# B&R Automation Studio project Soiled_PLC (part 18)

#### 16_sdc3Cyclic.ab
```automation-basic
PROGRAM _CYCLIC
	(* cyclic program *)

;Sequence 16 - Discharger 3 D[916]

;-----------------------------------------
;Revision 1.00 19/12/2005 D.J. First Issue
;-----------------------------------------

DischargerEnable 		= (NOT Std.HaltSys)

I_BagAtBuffer			= FALSE
I_BagAtDischarger		= X[8].X07
I_OpenBag				= X[8].X08
I_LoadDropped			= X[8].X08
I_BagReleased			= FALSE
I_BagEmpty			  	= TRUE

I_BagAtEmptyBuffer		= FALSE ;X[11].X07
O_EmptyBagBufferOpen	= FALSE ;Y[11].Y07

O_BagReady				= FALSE
O_OpenBuffer 			= FALSE
O_Steadys				= FALSE
O_Closer				= FALSE
O_OpenBag				= FALSE
O_OpenStop				= FALSE

;Enable.SDC[1]			= FALSE
Request.SDC[3]			= FALSE

;Alarm
Alarm[16].Name 			= almNoAlarm ;Clear sequence alarm name
Alarm[16].Bag 			= 263
Alarm[16].Beacon		= TRUE
Alarm[16].Extra			= 0
Alarm[16].Time			= 3000

;Setup Sequence
STEP = D[916]
;Setup Pulse contact
PLS = (STEP <> LASTSTEP)
LASTSTEP = STEP

;Step 0 - Disabled
IF (STEP = 0) THEN
	;Disabled
ENDIF

;Check Status - Bag settled at buffer, no bag at discharger, bag at buffer on screen and no bag at discharger on the screen
TON_10ms(I_BagAtBuffer,300,SettledAtBuffer,SettledAtBufferET)
IF (STEP = 1) THEN
	;IF (DischargerEnable AND SettledAtBuffer AND NOT I_BagAtDischarger AND (Bag[261].Cat > 0) AND (Bag[263].Cat = 0) AND NOT Std.HaltSys) THEN
	IF (DischargerEnable AND NOT I_BagAtDischarger AND (Bag[263].Cat = 0) AND NOT Std.HaltSys) THEN
		D[916] = 2
	ENDIF
	IF (Bag[263].Cat > 0) THEN
		Alarm[16].Name = almBagDataError
	ELSE IF I_BagAtDischarger THEN
		Alarm[16].Name = almSwitchFault
	;ELSE IF (Bag[263].Cat > 0) AND NOT I_BagAtBuffer THEN
	;	Alarm[16].Name 	= almBagDataError
	;	Alarm[16].Bag	= 263
	;ELSE IF (Bag[261].Cat = 0) AND I_BagAtBuffer THEN
	;	Alarm[16].Name 	= almBagNotShownOnScreen
	;	Alarm[16].Bag	= 261
	ENDIF
ENDIF

;Wait for bag in discharger
IF (STEP = 2) THEN
	;Enable.SDC[1]	= TRUE
	;O_OpenBuffer 	= TRUE
	IF I_BagAtDischarger THEN
		D[916] = 3
	ENDIF
	;Alarm[16].Name = almBagNotArrived
ENDIF

;Let bag settle in discharger
TON_10ms(((STEP = 3) AND I_BagAtDischarger),1000,SettledAtDischarger,SettledAtDischargerET)
IF (STEP = 3) THEN
	IF PLS  AND (Bag[263].Cat = 0) AND (Bag[252].Cat > 0) THEN
		Bag[252].Dst = 0
		Bag[263]     = Bag[252]
		Bag[252]     = Bag[0]
	ENDIF
	IF SettledAtDischarger THEN
		D[916] = 4
	ENDIF
	IF (Bag[263].Cat = Std.MaxCats) THEN
		D[916] = 11
	ENDIF
	Alarm[16].Name = almBagNotSettled
ENDIF

;Allow steadys to move down
TON_10ms((STEP = 4),400,SteadysDown,SteadysDownET)
IF (STEP = 4) THEN
	IF (SteadysDown AND NOT I_OpenBag) THEN
		D[916] = 5
	ENDIF
	IF I_OpenBag THEN
		Alarm[16].Name = almSwitchFault
	ENDIF
ENDIF

;Steady cylinders on from steps 4 - 9
O_Steadys = ((STEP >= 4) AND (STEP <= 9))

;Bag opener on from step 5 - 8
O_OpenBag = ((STEP >= 6) AND (STEP <= 8))

;Bag Ready to Washing Machine
IF (STEP = 5) THEN
	O_BagReady = TRUE
	IF I_OpenBag OR TestDischarger THEN
		D[916] = 6
	ENDIF
ENDIF

;Set LoadDropped to False
IF (STEP <> 6) THEN
	LoadDropped = FALSE
ENDIF

;Open Bag Until LoadDropped recieved and has been open for 6 seconds
TON_10ms((STEP = 6),600,MinOpen,MinOpenET) ;ET means Elapsed Time
IF (STEP = 6) THEN

	IF NOT I_OpenBag OR TestDischarger THEN
	;IF I_BagEmpty THEN
		LoadDropped = TRUE
	ENDIF

	IF (LoadDropped AND MinOpen) THEN
		;Write Report
		;------------
		IF (ReportUnloading[3].Cat = 0) THEN
			ReportUnloading[3].Cat = UINT(Bag[263].Cat)	;Category
			ReportUnloading[3].Cus = Bag[263].Cus		;Customer
			ReportUnloading[3].Wgt = Bag[263].Wgt		;Weight
			ReportUnloading[3].Cnt = 0					;Count
			ReportUnloading[3].Stn = 0					;Station
			ReportUnloading[3].Mcn = 3					;Machine
		ENDIF
	ENDIF
	IF (LoadDropped AND MinOpen) THEN
		D[916] = 7
	ENDIF
	Alarm[16].Name = almLoadNotDropped
ENDIF

;Change display to empty bag
IF (STEP = 7) THEN
	O_BagReady = Std.Clock500ms
	IF (I_OpenBag OR TestDrop) THEN
		Bag[263].Cat 	= Std.MaxCats
		D[916] 			= 8
	ENDIF
	Alarm[16].Name = almGeneralSequence
ENDIF

;Close bag
TON_10ms((STEP = 8),700,CloserDown,CloserDownET)
IF (STEP = 8) THEN
	O_Closer = TRUE
	IF CloserDown THEN
		D[916] = 9
	ENDIF
ENDIF

;Allow closer to go back up
TON_10ms((STEP = 9),700,CloserUp,CloserUpET)
IF (STEP = 9) THEN
	IF CloserUp THEN
		D[916] = 10
	ENDIF
ENDIF

;Allow steadys to go up
TON_10ms((STEP = 10),400,SteadyUp,SteadyUpET)
IF (STEP = 10) THEN
	IF SteadyUp THEN
		D[916] = 11
	ENDIF
ENDIF

;Check for space on empty bag buffer
IF (STEP = 11) THEN
	Request.SDC[3] = TRUE
	IF Enable.SDC[3] THEN
		D[916] = 12
	ENDIF
ENDIF

;Open buffer stop - unitl bag out
IF (STEP = 12) THEN
	O_OpenStop 	= TRUE
	Bag[263] 	= Bag[0]
	IF NOT Enable.SDC[3] THEN
		D[916] = 1
	ENDIF
	Alarm[16].Name = almBagNotReleased
ENDIF

;Alarms
TimerAlarm.IN 	= NOT PLS AND (Alarm[16].Name > 0)
TimerAlarm.PT 	= Alarm[16].Time
TimerAlarm FUB TON_10ms()
Alarm[16].On 	= TimerAlarm.Q
Alarm[16].ET 	= TimerAlarm.ET

;Outputs
Y[8].Y08 	= O_BagReady
;Y[6].Y01 	= O_OpenBuffer
Y[8].Y09 	= O_Steadys
Y[8].Y10 	= O_OpenBag
Y[8].Y05 	= O_Closer
Y[8].Y11 	= O_OpenStop
END_PROGRAM
```

### Program Logical/ExportsFromOriginal/17_svc2 (IEC, version 1.00.0) - * SVC2 Vertical Conveyor

#### 17_svc2Cyclic.ab
```automation-basic
PROGRAM _CYCLIC
	(* cyclic program *)

;---------------------------------------------------
;Sequence 13 - SIC2 Soiled Incline Conveyor 2 D[913]
;---------------------------------------------------

;Inputs
I_CarriageAtTop         = X[5].X02
I_CarriageAtBottom      = X[5].X03
I_BagOutAtTopSVC2       = X[7].X07
I_BagOutAtBottom		= X[4].X16
I_BagOnCarriageSVC2 	= X[5].X04
I_BagAtSVCBuffer        = X[6].X01

O_OpenCarriageStop		= FALSE
O_MoveUp 				= FALSE
O_MoveDown              = FALSE
O_BufferStop            = FALSE

Request.SVC[2] 			= FALSE

Alarm[17].Name 			= 0
Alarm[17].Bag			= 250
Alarm[17].Beacon		= TRUE
Alarm[17].Extra			= 0
Alarm[17].Time			= 3000

;Setup Sequence
STEP = D[917]
;Setup Pulse contact
PLS = (STEP <> LASTSTEP)
LASTSTEP = STEP

;Sequence
;Step 0 - Disabled
IF (STEP = 0) THEN
	;Disabled
ENDIF

;Move carriage up
IF (STEP = 1) THEN
	O_MoveUp = TRUE
	IF I_CarriageAtTop THEN
		D[917] = 2
	ENDIF
	IF NOT Std.EStop THEN
		Alarm[17].Name = almCarriageMoveFault
	ENDIF
ENDIF

;check carriage

IF (STEP = 2) THEN
	IF (NOT I_BagOnCarriageSVC2 AND NOT I_BagOutAtTopSVC2 AND  (Bag[250].Cat = 0) AND NOT Std.HaltSys) THEN

		D[917] = 3
	ENDIF
	IF (Bag[250].Cat > 0)  THEN
		Alarm[17].Name 	= almBagDataError
		Alarm[17].Bag	= 250
	ELSE IF  I_BagOnCarriage THEN
		Alarm[17].Name 	= almSwitchFault
		Alarm[17].Bag	= 250
	ENDIF
ENDIF

;request a bag
IF (STEP = 3) THEN
	;Request.SVC[2]  	= (I_CarriageAtTop AND NOT I_BagOnCarriageSVC2)
ENDIF

;Request a bag
TON_10ms(I_BagAtSVCBuffer AND (Bag[230].Cat > 0),200,BagAtBuffer,BagAtBufferET)
IF (STEP = 3) THEN

	IF (BagAtBuffer AND (Bag[230].Dst = 23) and (Bag[252].Cat = 0) and (Bag[263].Cat = 0) AND (D[916] = 2)) THEN
		D[917] = 4
	ELSE IF BagAtBuffer AND (Bag[230].Dst < 23) THEN
		D[917] = 4
	ENDIF

ENDIF

;wait for bag to arrive

IF (STEP = 4) THEN
	O_BufferStop  = TRUE

	IF (Bag[230].Dst = 23) AND I_CarriageAtTop   THEN
		O_OpenCarriageStop = TRUE
	ENDIF

	IF I_BagOutAtTopSVC2 AND O_OpenCarriageStop THEN
		IF((Bag[230].Cat > 0 ) AND (Bag[252].Cat = 0)) THEN
			Bag[252] = Bag[230]
			Bag[230] = Bag[0]
		ENDIF
		D[917] = 1
	ELSE IF ((Bag[230].Dst < 23) AND (Bag[230].Cat > 0)) THEN
		IF I_BagOnCarriageSVC2 THEN
			IF((Bag[230].Cat > 0 ) AND (Bag[250].Cat = 0)) THEN
				Bag[250] = Bag[230]
				Bag[230] = Bag[0]
			ENDIF
			D[917] = 5
		ENDIF

	ENDIF
ENDIF

;Allow bag to settle
TON_10ms(((STEP = 5) AND I_BagOnCarriageSVC2),300,BagSettled,BagSettledET)
IF (STEP = 5) THEN

	IF BagSettled THEN
		D[917] = 6
	ENDIF
	Alarm[17].Name = almBagNotSettled
ENDIF

;check bottom roller switch
IF (STEP = 6) THEN
	IF NOT I_CarriageAtBottom THEN
		D[917] = 7
	ENDIF
ENDIF

;move carriage down
IF (STEP = 7) THEN
	O_MoveDown 		= TRUE
	IF I_CarriageAtBottom THEN
		D[917] = 8
	ENDIF
ENDIF

;Check buffer has space
IF (STEP = 8) THEN
	IF Line[25].Clear AND (Bag[251].Cat = 0) AND (Bag[258].Cat = 0) AND NOT I_BagOutAtBottom THEN
		C[16] = 0
		C[25] = 0
		D[917] = 9
	ENDIF
	IF (Bag[258].Cat = 0) AND NOT Line[25].Clear THEN
		Alarm[17].Name = almBagNotSettled
		Alarm[17].Bag  = 258
	ENDIF
ENDIF

;Release bag low level

IF (STEP = 9) THEN
	O_OpenCarriageStop		= TRUE
	IF PLS THEN
		C[16] = 0
	ENDIF
	IF Line[16].Clear AND NOT PLS AND Carrstoptimer THEN
		IF ((Bag[250].Cat > 0) AND (Bag[251].Cat = 0)) THEN
			Bag[251] = Bag[250]
			Bag[250] = Bag[0]
		ENDIF
		D[917] = 10
	ENDIF
	Alarm[17].Name = almBagNotReleased
	Alarm[17].Bag  = 250
ENDIF
TON_10ms(((STEP = 9) AND O_OpenCarriageStop),750,Carrstoptimer,CarrstoptimerET)

;Bag at buffer stop high level
IF (STEP = 10) THEN
	IF BagAtBuffer THEN
		D[917] = 1
	ENDIF
ENDIF

;move trans bag to buffer
IF Line[25].Trip THEN
	IF ((Bag[251].Cat > 0) AND (Bag[258].Cat = 0)) THEN
		Bag[258] = Bag[251]
		Bag[251] = Bag[0]
	ENDIF
ENDIF

;Alarms
TimerAlarm.IN 	= NOT PLS AND (Alarm[17].Name > 0)
TimerAlarm.PT 	= Alarm[17].Time
TimerAlarm FUB TON_10ms()
Alarm[17].On 	= TimerAlarm.Q
Alarm[17].ET 	= TimerAlarm.ET

;Outputs

Y[9].Y03 =  (O_OpenCarriageStop	AND (I_CarriageAtTop OR I_CarriageAtBottom))
Y[9].Y01 =  (O_MoveUp AND NOT I_CarriageAtTop)
Y[9].Y02 =  (O_MoveDown AND NOT I_CarriageAtBottom)
Y[6].Y01 =  (O_BufferStop AND I_CarriageAtTop)
END_PROGRAM
```

#### 17_svc2.var
```iecst
VAR RETAIN
	STEP	:UINT;
	PLS	:BOOL;
	LASTSTEP	:UINT;
	O_OpenBufferStop	:BOOL;
	I_BagAtBuffer	:BOOL;
	O_RunMotor	:BOOL;
	BagSettled	:BOOL;
	BagSettledET	:TIME;
	BagAtBuffer	:BOOL;
	RunOnET	:TIME;
	RunOn	:BOOL;
	BagNearTopET	:TIME;
	BagNearTop	:BOOL;
	BagAtBufferET	:UDINT;
	I_BagInIncline	:BOOL;
END_VAR

VAR
	I_BagAtOutgoingBuffer	:BOOL;
	I_PaddleInPosition	:BOOL;
	CloseBufferStop	:BOOL;
	CloseBufferStopET	:TIME;
	O_OutgoingBufferOpen	:BOOL;
	TimerAlarm	:TON_10ms;
	O_SelectSP4ToSP2	:BOOL;
	I_BagReleased	:BOOL;
	O_SelectSP4	:BOOL;
	I_BagOutAtTop	:BOOL;
	I_BagOutAtBottom	:BOOL;
	I_BagOnCarriage	:BOOL;
	I_CarriageAtTop	:BOOL;
	I_CarriageAtBottom	:BOOL;
	O_OpenCarriageStop	:BOOL;
	O_MoveUp	:BOOL;
	O_MoveDown	:BOOL;
	I_BagAtSVCBuffer	:BOOL;
	O_BufferStop	:BOOL;
	Carrstoptimer	:BOOL;
	CarrstoptimerET	:TIME;
END_VAR
```

- Visualisation Logical/ExportsFromOriginal/svc1 (not shown)

### Data object Logical/ExportsFromOriginal/can_cmd (Simple) - * Powertrans 1 & 2

#### can_cmd.dat
```
;-----------------
;CAN Command Table
;-----------------

;         1234567890123456789012345678901   1234567890123456789012345678901
00000121,"ReadFrame1                     ","EventRead1                     ",$00000000
00000120,"WriteFrame1                    ","EventWrite1                    ",$00000001

00000131,"ReadFrame2                     ","EventRead2                     ",$00000000
00000130,"WriteFrame2                    ","EventWrite2                    ",$00000001

;00000141,"ReadFrame3                     ","EventRead3                     ",$00000000
;00000140,"WriteFrame3                    ","EventWrite3                    ",$00000001
;   |          |                                 |                               |
; CAN ADR  Variable Name 31 Chrs             Event Variable 31 Chrs           Read = 0 Write = 1
```

### Program Logical/ExportsFromOriginal/can_drv2 (IEC, version 1.00.0) - * PowerTrans 1 SDC2

#### can_drv2Cyclic.ab
```automation-basic
PROGRAM _CYCLIC
;----------------------------------------
;Version 1.00 08/02/2005 D.J. First Issue
;----------------------------------------

IF CANOK THEN

	;----------------
	;Set Write values
	;----------------

	;Powertrans 1
	IF CAN[1].BagReady THEN
		WriteFrame1.ControlSignals = BIT_SET(WriteFrame1.ControlSignals, 1)
	ELSE
		WriteFrame1.ControlSignals = BIT_CLR(WriteFrame1.ControlSignals, 1)
	ENDIF
	;IF CAN[1].DoubleLoad THEN
	;	WriteFrame1.ControlSignals = BIT_SET(WriteFrame1.ControlSignals, 2)
	;ELSE
	;	WriteFrame1.ControlSignals = BIT_CLR(WriteFrame1.ControlSignals, 2)
	;ENDIF
	WriteFrame1.Destination = 0
	WriteFrame1.Category 	= CAN[1].Category
	WriteFrame1.Customer    = CAN[1].Customer
	WriteFrame1.Weight      = CAN[1].Weight

	;Write to Machine1
	EventWrite1 = TRUE

	;Powertrans 2
	IF CAN[2].BagReady THEN
		WriteFrame2.ControlSignals = BIT_SET(WriteFrame2.ControlSignals, 1)
	ELSE
		WriteFrame2.ControlSignals = BIT_CLR(WriteFrame2.ControlSignals, 1)
	ENDIF
	;IF CAN[2].DoubleLoad THEN
	;	WriteFrame2.ControlSignals = BIT_SET(WriteFrame2.ControlSignals, 2)
	;ELSE
	;	WriteFrame2.ControlSignals = BIT_CLR(WriteFrame2.ControlSignals, 2)
	;ENDIF
	WriteFrame2.Destination = 0
	WriteFrame2.Category 	= CAN[2].Category
	WriteFrame2.Customer    = CAN[2].Customer
	WriteFrame2.Weight      = CAN[2].Weight

	;Write to Machine2
	EventWrite2 = TRUE

	;-----------------
	;Service CAN table
	;-----------------

	IF CANdftab_01.status=0 THEN						(*check error level*)
		CANrwtab_01.enable		= 1
		CANrwtab_01.tab_ident	= CANdftab_01.tab_ident (*define tab_id*)
		CANrwtab_01 FUB CANrwtab()						(*initiate CANrwtab*)
		LastError = CANrwtab_01.status
	ENDIF

	;----------------------------------
	;Check for incomming data from CBW1
	;----------------------------------

	;Powertrans 1
	IF EventRead1 THEN

		EventRead1 = FALSE

		CAN[1].Live 		  = BIT_TST(ReadFrame1.ControlSignals,0)
		CAN[1].DropLoad 	  = BIT_TST(ReadFrame1.ControlSignals,1)
		CAN[1].LoadDropped    = BIT_TST(ReadFrame1.ControlSignals,2)

		IF CAN[1].Live THEN
			CAN[1].LiveTime = 50	;5 seconds
		ENDIF

	ENDIF

	;----------------------------------
	;Check for incomming data from CBW2
	;----------------------------------

	;Powertrans 2
	IF EventRead2 THEN

		EventRead2 = FALSE

		CAN[2].Live 		  = BIT_TST(ReadFrame2.ControlSignals,0)
		CAN[2].DropLoad 	  = BIT_TST(ReadFrame2.ControlSignals,1)
		CAN[2].LoadDropped    = BIT_TST(ReadFrame2.ControlSignals,2)

		IF CAN[2].Live THEN
			CAN[2].LiveTime = 50	;5 seconds
		ENDIF

	ENDIF

	;-------------------
	;CAN Live / Presence
	;-------------------

	LOOP n = 1 TO 2 DO

		IF (CAN[n].LiveTime > 0) THEN
			CAN[n].LiveTime = (CAN[n].LiveTime - 1)
		ENDIF

		CAN[n].Live = (CAN[n].LiveTime <> 0)

	ENDLOOP

ENDIF
END_PROGRAM
```

#### can_drv2Init.ab
```automation-basic
PROGRAM _INIT
	(* init program *)

CAN_enable = 1
EventWrite1 = 0									;Reset CAN data table WRITE event
EventRead1 = 0  								;Reset CAN data table READ event
;EventWrite2 = 0								;Reset CAN data table WRITE event
;EventRead2 = 0  								;Reset CAN data table READ event
;EventWrite3 = 0								;Reset CAN data table WRITE event
;EventRead3 = 0  							    ;Reset CAN data table READ event

CANopen_01.enable		= CAN_enable
CANopen_01.baud_rate	= 25					;Define baud rate - 250 kbit/s
CANopen_01.cob_anz		= 100      				;Define number of link objects
CANopen_01.error_adr	= ADR(error_var)		;Define address for error output
CANopen_01.device		= ADR("SS1.IF2")	;Define number of device
CANopen_01.info			= 0

CANopen_01 FUB CANopen()						;Initiate CANopen

IF CANopen_01.status=0 THEN						;Check error level

	DOInfo.enable = 1
	DOInfo.pName  = "can_cmd"

	DOInfo FUB DatObjInfo()

	IF (DOInfo.status = 0) THEN

		data_adr					= DOInfo.pDatObjMem
		CANdftab_01.enable			= 1
		CANdftab_01.us_ident 		= CANopen_01.us_ident	;Set us_id
		CANdftab_01.table_adr		= data_adr				;Define address of data object
		CANdftab_01.tab_num			= UINT(DOInfo.len / 72)	;Define number of values

		CANdftab_01 FUB CANdftab()    						;Initiate CANdftab

		IF CANdftab_01.status = 0 THEN
			WriteFrame1.ControlSignals = BIT_SET(WriteFrame1.ControlSignals,0);Set Live Signal
			WriteFrame2.ControlSignals = BIT_SET(WriteFrame2.ControlSignals,0)
			;WriteFrame3.ControlSignals = BIT_SET(WriteFrame3.ControlSignals,0)
			CANOK = TRUE
		ENDIF

	ENDIF

ENDIF
END_PROGRAM
```

#### can_drv2.var
```iecst
VAR RETAIN
	CAN_enable	:BOOL;
	ReadFrame1	:WET_CAN;
	EventRead1	:BOOL;
	EventWrite1	:BOOL;
	LastError	:UINT;
	n	:UINT;
	CANOK	:BOOL;
	WriteFrame1	:WET_CAN;
	EventWrite2	:BOOL;
END_VAR

VAR
	ReadFrame2	:WET_CAN;
	EventRead2	:BOOL;
	WriteFrame2	:WET_CAN;
	CANopen_01	:CANopen;
	DOInfo	:DatObjInfo;
	CANdftab_01	:CANdftab;
	error_var	:UDINT;
	data_adr	:UDINT;
	CANrwtab_01	:CANrwtab;
END_VAR
```

### Program Logical/ExportsFromOriginal/can_dis (IEC, version 1.00.0)

#### can_disCyclic.ab
```automation-basic
PROGRAM _CYCLIC
;-----------------------------------------
;Revision 1.00 18/02/2002 D.J. First Issue
;-----------------------------------------

;2 * 20 or 2 * 40 chr VFD display

;Set D register where text for display is set E register for weight
DisplayChrs		= 80

LOOP m = 1 TO 16 DO
	DisplayCat[m] = (4000 + ((m - 1) * 80))
	DisplayCus[m] = DisplayCat[m] + 40
	DisplayWgt[m] = Bag[200 + m].Wgt
ENDLOOP

LOOP x = 1 to 16 DO

	memcpy(ADR(Display[0]) ,ADR(D[DisplayCat[x]]),DisplayChrs)
	memcpy(ADR(Display[44]),ADR(D[DisplayCus[x]]),DisplayChrs)

	;As the weight value is a INT put into a UINT -0.1 = 65535
	;Display only if less than 500kg
	IF (DisplayWgt[x] < 5000) THEN
		DIS4(DisplayWgt[x],TRUE,Dummy,Wgt1s,Wgt10s,Dummy)
	ELSE
		Wgt1s 	= 0
		Wgt10s 	= 0
	ENDIF

	;Add Weight and goto next line
	Display[35] = $20 ;Space
	Display[36] = (48 + USINT(Wgt10s))
	Display[37] = (48 + USINT(Wgt1s))
	Display[38] = $6B 	;k
	Display[39] = $67 	;g
	Display[40] = $A	;Line Feed
	Display[41] = $D	;Carriage Return
	Display[42] = 0
	Display[43] = 0

	;Display[78] = $44	;D
	;Display[79] = $55	;U
	;Display[80] = $43	;C
	;Display[81] = $4B	;K
	;Display[82] = $45	;E
	;Display[83] = $52	;R

	;Cursor Off and Home
	IF (STEP = 0) THEN
		n = 0
		Data.Data[0] = $9B
		Data.Data[1] = $6C
		Data.Data[2] = $9B
		Data.Data[3] = $48
		Data.Data[4] = 0
		Data.Data[5] = 0
		Data.Data[6] = 0
		Data.Data[7] = 0
	ENDIF

	;Write text to the Display
	IF (STEP > 0) THEN
		Data.Data[0] = USINT(Display[0 + n])
		Data.Data[1] = USINT(Display[1 + n])
		Data.Data[2] = USINT(Display[2 + n])
		Data.Data[3] = USINT(Display[3 + n])
		Data.Data[4] = USINT(Display[4 + n])
		Data.Data[5] = USINT(Display[5 + n])
		Data.Data[6] = USINT(Display[6 + n])
		Data.Data[7] = USINT(Display[7 + n])
	ENDIF

	;Write to the CAN Frame For the Current Display
	IF (x = 1) THEN
		DisplayTXFrame1 = Data
	ELSE IF (x = 2) THEN
		DisplayTXFrame2 = Data
	ELSE IF (x = 3) THEN
		DisplayTXFrame3 = Data
	ELSE IF (x = 4) THEN
		DisplayTXFrame4 = Data
	ELSE IF (x = 5) THEN
		DisplayTXFrame5 = Data
	ELSE IF (x = 6) THEN
		DisplayTXFrame6 = Data
	ELSE IF (x = 7) THEN
		DisplayTXFrame7 = Data
	ELSE IF (x = 8) THEN
		DisplayTXFrame8 = Data
	ELSE IF (x = 9) THEN
		DisplayTXFrame9 = Data
	ELSE IF (x = 10) THEN
		DisplayTXFrame10 = Data
	ELSE IF (x = 11) THEN
		DisplayTXFrame11 = Data
	ELSE IF (x = 12) THEN
		DisplayTXFrame12 = Data
	ELSE IF (x = 13) THEN
		DisplayTXFrame13 = Data
	ELSE IF (x = 14) THEN
		DisplayTXFrame14 = Data
	ELSE IF (x = 15) THEN
		DisplayTXFrame15 = Data
	ELSE IF (x = 16) THEN
		DisplayTXFrame16 = Data
	ENDIF

ENDLOOP

IF (STEP > 0) THEN
	n = n + 8
ENDIF

STEP = STEP + 1

StepsRequired = ((DisplayChrs / 8) + 1) ;Steps = Total Chrs / 8 + 1
IF STEP > StepsRequired THEN
	STEP = 0
ENDIF

IF CANOK THEN

	;------------------------------------------------------
	;Configure the CAN write to CBW1 SDC1
	;------------------------------------------------------

	;Write to Displays
	DisplayWrite1 = TRUE
	;DisplayWrite2 = TRUE
	DisplayWrite3 = TRUE
	;DisplayWrite4 = TRUE
	DisplayWrite5 = TRUE
	;DisplayWrite6 = TRUE
	DisplayWrite7 = TRUE
	;DisplayWrite8 = TRUE
	;DisplayWrite9 = TRUE
	;DisplayWrite10 = TRUE
	;DisplayWrite11 = TRUE
	;DisplayWrite12 = TRUE
	;DisplayWrite13 = TRUE
	;DisplayWrite14 = TRUE
	;DisplayWrite15 = TRUE
	;DisplayWrite16 = TRUE

	;------------------------
	;Service CAN table
	;------------------------

	IF CANdftab_01.status=0 THEN						(*check error level*)
		CANrwtab_01.enable		= 1
		CANrwtab_01.tab_ident	= CANdftab_01.tab_ident (*define tab_id*)
		CANrwtab_01 FUB CANrwtab()						(*initiate CANrwtab*)
		LastError = CANrwtab_01.status
	ENDIF

	;-----------------
	;Read Display Data
	;-----------------
	IF DisplayRead1 THEN
		DisplayRead1 = FALSE
		Reply = DisplayRXFrame1.Data[1]
	ENDIF
	IF DisplayRead2 THEN
		DisplayRead2 = FALSE
		Reply = DisplayRXFrame2.Data[1]
	ENDIF
	IF DisplayRead3 THEN
		DisplayRead3 = FALSE
		Reply = DisplayRXFrame3.Data[1]
	ENDIF
	IF DisplayRead4 THEN
		DisplayRead4 = FALSE
		Reply = DisplayRXFrame4.Data[1]
	ENDIF
	IF DisplayRead5 THEN
		DisplayRead5 = FALSE
		Reply = DisplayRXFrame5.Data[1]
	ENDIF
	IF DisplayRead6 THEN
		DisplayRead6 = FALSE
		Reply = DisplayRXFrame6.Data[1]
	ENDIF
	IF DisplayRead7 THEN
		DisplayRead7 = FALSE
		Reply = DisplayRXFrame7.Data[1]
	ENDIF
	IF DisplayRead8 THEN
		DisplayRead8 = FALSE
		Reply = DisplayRXFrame8.Data[1]
	ENDIF
	IF DisplayRead9 THEN
		DisplayRead9 = FALSE
		Reply = DisplayRXFrame9.Data[1]
	ENDIF
	IF DisplayRead10 THEN
		DisplayRead10 = FALSE
		Reply = DisplayRXFrame10.Data[1]
	ENDIF
	IF DisplayRead11 THEN
		DisplayRead11 = FALSE
		Reply = DisplayRXFrame11.Data[1]
	ENDIF
	IF DisplayRead12 THEN
		DisplayRead12 = FALSE
		Reply = DisplayRXFrame12.Data[1]
	ENDIF
	IF DisplayRead13 THEN
		DisplayRead13 = FALSE
		Reply = DisplayRXFrame13.Data[1]
	ENDIF
	IF DisplayRead14 THEN
		DisplayRead14 = FALSE
		Reply = DisplayRXFrame14.Data[1]
	ENDIF
	IF DisplayRead15 THEN
		DisplayRead15 = FALSE
		Reply = DisplayRXFrame15.Data[1]
	ENDIF
	IF DisplayRead16 THEN
		DisplayRead16 = FALSE
		Reply = DisplayRXFrame16.Data[1]
	ENDIF

ENDIF
END_PROGRAM
```

#### can_disInit.ab
```automation-basic
PROGRAM _INIT
	(* init program *)

CAN_enable = 1
DisplayWrite1 = 0								;Reset CAN data table WRITE event
DisplayRead1 = 0  								;Reset CAN data table READ event
;EventWrite2 = 0								;Reset CAN data table WRITE event
;EventRead2 = 0  								;Reset CAN data table READ event
;EventWrite3 = 0								;Reset CAN data table WRITE event
;EventRead3 = 0  							    ;Reset CAN data table READ event

CANopen_01.enable		= CAN_enable
CANopen_01.baud_rate	= 25					;Define baud rate - 250 kbit/s
CANopen_01.cob_anz		= 100      				;Define number of link objects
CANopen_01.error_adr	= ADR(error_var)		;Define address for error output
CANopen_01.device		= ADR("SS1.IF3")		;Define number of device
CANopen_01.info			= 0

CANopen_01 FUB CANopen()						;Initiate CANopen

IF CANopen_01.status=0 THEN						;Check error level

	DOInfo.enable = 1
	DOInfo.pName  = "disp_cmd"

	DOInfo FUB DatObjInfo()

	IF (DOInfo.status = 0) THEN

		data_adr					= DOInfo.pDatObjMem
		CANdftab_01.enable			= 1
		CANdftab_01.us_ident 		= CANopen_01.us_ident	;Set us_id
		CANdftab_01.table_adr		= data_adr				;Define address of data object
		CANdftab_01.tab_num			= UINT(DOInfo.len / 72)	;Define number of values

		CANdftab_01 FUB CANdftab()    						;Initiate CANdftab

		IF CANdftab_01.status = 0 THEN
			CANOK = TRUE
		ENDIF

	ENDIF

ENDIF
END_PROGRAM
```

#### can_dis.var
```iecst
VAR RETAIN
	CAN_enable	:BOOL;
	LastError	:UINT;
	n	:UINT;
	CANOK	:BOOL;
END_VAR

VAR
	CANopen_01	:CANopen;
	DOInfo	:DatObjInfo;
	CANdftab_01	:CANdftab;
	error_var	:UDINT;
	data_adr	:UDINT;
	CANrwtab_01	:CANrwtab;
	DisplayWrite1	:BOOL;
	DisplayRead1	:BOOL;
	DisplayCat	:ARRAY [0..16] OF UINT;
	DisplayWgt	:ARRAY [0..12] OF UINT;
	DisplayCus	:ARRAY [0..16] OF UINT;
	Display	:ARRAY [0..87] OF UINT;
	Data	:WriteDisplay;
	Reply	:USINT;
	DisplayRXFrame5	:ReadDisplay;
	DisplayRXFrame4	:ReadDisplay;
	DisplayWrite4	:BOOL;
	DisplayTXFrame1	:WriteDisplay;
	DisplayWrite5	:BOOL;
	DisplayTXFrame2	:WriteDisplay;
	x	:UINT;
	DisplayWrite6	:BOOL;
	DisplayTXFrame3	:WriteDisplay;
	DisplayRead2	:BOOL;
	DisplayTXFrame4	:WriteDisplay;
	DisplayRead3	:BOOL;
	DisplayTXFrame5	:WriteDisplay;
	Dummy	:UINT;
	DisplayRead4	:BOOL;
	DisplayRXFrame1	:ReadDisplay;
	DisplayTXFrame6	:WriteDisplay;
	DisplayRead5	:BOOL;
	DisplayRXFrame2	:ReadDisplay;
	DisplayRead6	:BOOL;
	DisplayRXFrame3	:ReadDisplay;
	StepsRequired	:UINT;
	DisplayChrs	:UINT;
	DisplayRXFrame6	:ReadDisplay;
	STEP	:UINT;
	Wgt1s	:UINT;
	DisplayWrite2	:BOOL;
	DisplayWrite3	:BOOL;
	Wgt10s	:UINT;
	m	:UINT;
	DisplayTXFrame7	:WriteDisplay;
	DisplayTXFrame8	:WriteDisplay;
	DisplayTXFrame9	:WriteDisplay;
	DisplayTXFrame10	:WriteDisplay;
	DisplayTXFrame11	:WriteDisplay;
	DisplayTXFrame12	:WriteDisplay;
	DisplayTXFrame13	:WriteDisplay;
	DisplayWrite7	:BOOL;
	DisplayWrite8	:BOOL;
	DisplayWrite9	:BOOL;
	DisplayWrite10	:BOOL;
	DisplayWrite11	:BOOL;
	DisplayWrite12	:BOOL;
	DisplayWrite13	:BOOL;
	DisplayWrite14	:BOOL;
	DisplayWrite15	:BOOL;
	DisplayWrite16	:BOOL;
	DisplayRead7	:BOOL;
	DisplayRead8	:BOOL;
	DisplayRead9	:BOOL;
	DisplayRead10	:BOOL;
	DisplayRead11	:BOOL;
	DisplayRead12	:BOOL;
	DisplayRead13	:BOOL;
	DisplayRead14	:BOOL;
	DisplayRead15	:BOOL;
	DisplayRead16	:BOOL;
	DisplayRXFrame7	:ReadDisplay;
	DisplayRXFrame8	:ReadDisplay;
	DisplayRXFrame9	:ReadDisplay;
	DisplayRXFrame10	:ReadDisplay;
	DisplayRXFrame11	:ReadDisplay;
	DisplayRXFrame12	:ReadDisplay;
	DisplayRXFrame13	:ReadDisplay;
	DisplayRXFrame14	:ReadDisplay;
	DisplayRXFrame15	:ReadDisplay;
	DisplayRXFrame16	:ReadDisplay;
	DisplayTXFrame14	:WriteDisplay;
	DisplayTXFrame15	:WriteDisplay;
	DisplayTXFrame16	:WriteDisplay;
END_VAR
```

### Data object Logical/ExportsFromOriginal/disp_cmd (Simple, version 1.00.0)

#### disp_cmd.dat
```
;-----------------
;CAN Command Table
;-----------------

;         1234567890123456789012345678901   1234567890123456789012345678901
;CAN Node 11
00001215,"DisplayRXFrame1                ","DisplayRead1                   ",$00000000
00001214,"DisplayTXFrame1                ","DisplayWrite1                  ",$00000001
;CAN Node 12
;00001231,"DisplayRXFrame2                ","DisplayRead2                   ",$00000000
;00001230,"DisplayTXFrame2                ","DisplayWrite2                  ",$00000001
;CAN Node 13
00001247,"DisplayRXFrame3                ","DisplayRead3                   ",$00000000
00001246,"DisplayTXFrame3                ","DisplayWrite3                  ",$00000001
;CAN Node 14
;00001263,"DisplayRXFrame4                ","DisplayRead4                   ",$00000000
;00001262,"DisplayTXFrame4                ","DisplayWrite4                  ",$00000001
;CAN Node 15
00001279,"DisplayRXFrame5                ","DisplayRead5                   ",$00000000
00001278,"DisplayTXFrame5                ","DisplayWrite5                  ",$00000001
;CAN Node 16
;00001295,"DisplayRXFrame6                ","DisplayRead6                   ",$00000000
;00001294,"DisplayTXFrame6                ","DisplayWrite6                  ",$00000001
;CAN Node 17
00001311,"DisplayRXFrame7                ","DisplayRead7                   ",$00000000
00001310,"DisplayTXFrame7                ","DisplayWrite7                  ",$00000001
;CAN Node 18
;00001327,"DisplayRXFrame8                ","DisplayRead8                   ",$00000000
;00001326,"DisplayTXFrame8                ","DisplayWrite8                  ",$00000001
;CAN Node 19
;00001343,"DisplayRXFrame9                ","DisplayRead9                   ",$00000000
;00001342,"DisplayTXFrame9                ","DisplayWrite9                  ",$00000001
;CAN Node 20
;00001359,"DisplayRXFrame10               ","DisplayRead10                  ",$00000000
;00001358,"DisplayTXFrame10               ","DisplayWrite10                 ",$00000001
;CAN Node 21
;00001375,"DisplayRXFrame11               ","DisplayRead11                  ",$00000000
;00001374,"DisplayTXFrame11               ","DisplayWrite11                 ",$00000001
;CAN Node 22
;00001391,"DisplayRXFrame12               ","DisplayRead12                  ",$00000000
;00001390,"DisplayTXFrame12               ","DisplayWrite12                 ",$00000001
;CAN Node 23
;00001407,"DisplayRXFrame13               ","DisplayRead13                  ",$00000000
;00001406,"DisplayTXFrame13               ","DisplayWrite13                 ",$00000001
;CAN Node 24
;00001423,"DisplayRXFrame14               ","DisplayRead14                  ",$00000000
;00001422,"DisplayTXFrame14               ","DisplayWrite14                 ",$00000001
;CAN Node 25
;00001439,"DisplayRXFrame15               ","DisplayRead15                  ",$00000000
;00001438,"DisplayTXFrame15               ","DisplayWrite15                 ",$00000001
;CAN Node 26
;00001455,"DisplayRXFrame16               ","DisplayRead16                  ",$00000000
;00001454,"DisplayTXFrame16               ","DisplayWrite16                 ",$00000001

;   |          |                                 |                               |
; CAN ADR  Variable Name 31 Chrs             Event Variable 31 Chrs           Read = 0 Write = 1
```

### Safety.typ
```iecst
TYPE
	SafeInterlockType : 	STRUCT
		GS_DI_01_Access_Reset : BOOL; (*Interlock access request and zone reset operator input*)
		GS_DI_02_Monitor_Solenoid : BOOL; (*Interlock solenoid feedback*)
		GS_DO_01_Lock_Solenoid : BOOL; (*Interlock solenoid output*)
		GS_Two_Channel_Input : BOOL; (*Safe PLC feedback of the state of interlock dual channel*)
	END_STRUCT;
	SafeE_StopType : 	STRUCT
		ES_SI_Two_Channel : ARRAY[0..MAX_DUAL_CHANNELS]OF BOOL; (*Safe PLC feedback of the state of e-stop dual channel*)
	END_STRUCT;
	SafeTowerLightType : 	STRUCT
		TL_DO_Green : BOOL; (*Tower light output for Green light*)
		TL_DO_Yellow : BOOL; (*Tower light output for Yellow light*)
		TL_DO_Red : BOOL; (*Tower light output for Red light*)
		TL_DO_Sounder : BOOL; (*Tower light output for sounder*)
	END_STRUCT;
	SafeZoneType : 	STRUCT
		Interlock : SafeInterlockType; (*Interlock structure*)
		E_Stop : SafeE_StopType; (*Emergency stop structure*)
		TowerLight : SafeTowerLightType; (*Tower light structure*)
		Zone_Status : BOOL; (*State of the zone passed back from safe PLC*)
		AccessRequested : BOOL; (*Operator as requested access*)
		BagsInTransit : BOOL; (*True = Sequences are still not in a safe step*)
		HoistsOutOfPosition : BOOL; (*True = Hoists in zone are not parked*)
		Main_Reset : BOOL; (*Main panel reset*)
		Main_Lamp : BOOL; (*Main panel lamp*)
		Disable : BOOL; (*Passed into sequences to inhibit stepping on*)
		EDM : BOOL; (*EDM Feedback from linking relays*)
		ResetReady : BOOL; (*Zone is ready to be reset*)
		LiftGates : BOOL; (*Lift the edge protection gates.*)
	END_STRUCT;
	Safety_Hoist_type : 	STRUCT
		I_Operator_PushButton : BOOL; (*Bulk loading operator push button*)
		O_OpenGuard : BOOL; (*Sliding guard output*)
		O_CloseGuard : BOOL; (*Sliding guard output*)
		OutOfPosition : BOOL; (*True when hoist is not in Service position*)
		I_GuardClosed : BOOL; (*Sliding guard closed*)
	END_STRUCT;
END_TYPE
```

### Safety.var
```iecst
VAR
	SafetyZone : ARRAY[0..MAX_SAFE_ZONES] OF SafeZoneType;
	Safety_Master_Reset : BOOL;
	Safety_Module_Fault : BOOL;
	Hoist_Safety : ARRAY[0..MAX_HOIST] OF Safety_Hoist_type;
END_VAR
VAR CONSTANT
	MAX_SAFE_ZONES : USINT := 3;
	MAX_DUAL_CHANNELS : USINT := 1;
	MAX_HOIST : USINT := 1;
END_VAR
```

### Program Logical/Safety/Safety (IEC, version 1.00.4)

#### Main.st - Safet Task must come after all task with gaurded areas
```iecst
//---------------------------------------------
//-------------Safety Request------------------
//---------------------------------------------
//V1.00.2 -- 2019 May 24 -- TR -- Fix issue with master reset not working if not ready.
//V1.00.3 -- 2019 June 26 -- TR -- FIx issue with the solenoid not opening if the hoist switch is made after the bagInTransit timers.. Add timer for hoist in position so the hoist cannot be moving past the safe position and open the door.
//V1.00.4 -- 2019 November 11 -- TR -- 	FIX: Issues with the solenoid locking incorrectly,
										//ADD: Control to lift the edge protection gates ( Map Directly to all required outputs.)
PROGRAM _INIT
debounceMasterPT := 200; //2 second
transitSettlePT := 3000; //3000seconds
startUpWarningPT := 500; //5 secs
enableMasterReset := TRUE; // Set to true if master reset is to be used
FOR n:=0 TO MAX_SAFE_ZONES DO
	safeState[n] := 4;
END_FOR;
END_PROGRAM

PROGRAM _CYCLIC

ton_10ms_startUp_Warning(IN:=ton_10ms_Master_Reset.Q, PT:=startUpWarningPT);
Safety_Master_Reset := ton_10ms_startUp_Warning.Q AND Std.Clock1s;

IF SafetyZone[0].Main_Reset AND enableMasterReset THEN
	masterResetRequest := 1; // Set masterResetRequest
END_IF;
ton_10ms_Master_Reset(IN:= masterResetRequest, PT:=debounceMasterPT);

FOR n:=0 TO MAX_SAFE_ZONES DO
	//-------------------------------------------------------
	//---------------------Master-reset----------------------
	//-------------------------------------------------------

	lockDoor[n] := FALSE;

	tof_HoistsOutOfPosition[n].IN := SafetyZone[n].HoistsOutOfPosition;
	tof_HoistsOutOfPosition[n].PT := 100;
	tof_HoistsOutOfPosition[n]();

	ton_entryError[n].IN := (safeState[n] = 3);
	ton_entryError[n].PT := 100;
	ton_entryError[n]();

	IF ton_10ms_Master_Reset.Q AND NOT SafetyZone[n].Zone_Status AND SafetyZone[n].ResetReady THEN // only put a zone to reset if it needs it
		masterReset[n] := TRUE; // Set masterReset
		safeState[n] := 10; // Goto master reset state
	END_IF;

	//-------------------------------------------------------
	//------------------END-Master-Reset-END-----------------
	//-------------------------------------------------------

	//-------------------------------------------------------
	//------------------Safety-State-Machine-----------------
	//-------------------------------------------------------

	//Wait for bags to finish moving and hoists to get into position.. Door can be unlocked
	ton_10ms_Transit_Settle[n](IN:=SafetyZone[n].AccessRequested AND (safeState[n] = 1), PT:=transitSettlePT);
	f_trigRequestAccess[n].CLK:= SafetyZone[n].Interlock.GS_DI_01_Access_Reset;
	f_trigRequestAccess[n]();
	CASE safeState[n] OF
		0: //Zone reset do not enter

			// Operator requests access by pressing Access DI for 1 second then releasing
			//ton_10ms_Access_Debounce[n](IN:=SafetyZone[n].Interlock.GS_DI_01_Access_Reset, PT:=debouncePT);
			//Request Access on f_trig of pressing reset. if the zone is healthy
			//SafetyZone[n].Interlock.GS_DO_01_Lock_Solenoid := FALSE; //Reset after reset pressed and door shut
			IF SafetyZone[n].Zone_Status AND f_trigRequestAccess[n].Q  THEN//	ELSIF (debounceEdgeNeg[n] OR SafetyZone[n].AccessRequested) AND NOT masterReset THEN //Look for falling edge if masterReset not requested
				SafetyZone[n].AccessRequested := TRUE; //Reset after unlocking or safe zone goes off
				safeState[n] := 1; //Access has been requested
				masterReset[n] := 0;
				//If zone accessed by override or depedant Zone drops out.
			ELSIF NOT SafetyZone[n].Zone_Status AND NOT SafetyZone[n].Interlock.GS_Two_Channel_Input THEN //If entered with overide goto state 3
				safeState[n] := 3;
			ELSIF NOT SafetyZone[n].Zone_Status AND SafetyZone[n].Interlock.GS_Two_Channel_Input THEN //If dependant zone drops out
				safeState[n] := 4;
			END_IF;

		1: //Access has been requested
			//Allow 1 second for moving bags to settle, once ok
			ton_10ms_bagsInTransit[n](IN:=NOT SafetyZone[n].BagsInTransit, PT:=100); //buffer the BagsInTransit bool

			//Latch solenoid lock open
			IF ton_10ms_bagsInTransit[n].Q AND SafetyZone[n].Disable AND NOT tof_HoistsOutOfPosition[n].Q THEN //Use Disable instead of AccessRequested, to ensure one cyclic check with Disable on to stop BagsInTransit being missed
				//SafetyZone[n].Interlock.GS_DO_01_Lock_Solenoid := TRUE; //Reset after reset pressed and door shut
				safeState[n] := 2; //Safe to enter no bags in transit
			ELSIF ton_10ms_Transit_Settle[n].Q THEN
				//SafetyZone[n].Interlock.GS_DO_01_Lock_Solenoid := NOT tof_HoistsOutOfPosition[n].Q; //Reset after reset pressed and door shut
				safeState[n] := 3; //Waiting time elapsed, enter with caution
			END_IF;

			//If zone accessed by override or depedant Zone drops out.
			IF NOT SafetyZone[n].Zone_Status AND NOT SafetyZone[n].Interlock.GS_Two_Channel_Input THEN //If entered with overide goto state 3
				safeState[n] := 3;
			ELSIF NOT SafetyZone[n].Zone_Status AND SafetyZone[n].Interlock.GS_Two_Channel_Input THEN //If dependant zone drops out
				safeState[n] := 4;
			ELSIF SafetyZone[n].Zone_Status AND f_trigRequestAccess[n].Q THEN //Cancel the request
				SafetyZone[n].AccessRequested := FALSE; //Reset after safe zone goes off
				safeState[n] := 4;
			END_IF;

		2..3: //Zone unlocked
			//Reset access request
			lockDoor[n] := NOT tof_HoistsOutOfPosition[n].Q;

			IF SafetyZone[n].AccessRequested AND NOT SafetyZone[n].Zone_Status THEN
				SafetyZone[n].AccessRequested := FALSE; //Reset after safe zone goes off
				IF n = 0 THEN
					safeState[n] := 0; //Zone reset do not enter
				END_IF
			ELSIF SafetyZone[n].Zone_Status AND f_trigRequestAccess[n].Q  AND SafetyZone[n].AccessRequested THEN //Cancel the request
				SafetyZone[n].AccessRequested := FALSE; //Reset after safe zone goes off
				safeState[n] := 4;
			ELSIF SafetyZone[n].Zone_Status AND NOT SafetyZone[n].AccessRequested THEN // zone has been accessed and reset.
				safeState[n] := 0;
			END_IF;

		4:
			//Reset tower light state only if safety plc feedback ok
			IF SafetyZone[n].Zone_Status THEN //Check Safe PLC status
				safeState[n] := 0; //Zone reset do not enter
			END_IF;

		10: // Master reset
			IF (SafetyZone[n].Zone_Status OR NOT SafetyZone[n].ResetReady) THEN
				safeState[n] := 0;
				masterReset[n] := FALSE;
			END_IF;

	END_CASE;

//	//Lock solenoid
//	//ton_10ms_Reset_Debounce[n](IN:=SafetyZone[n].Interlock.GS_DI_01_Access_Reset, PT:=debouncePT);
//	IF (SafetyZone[n].Interlock.GS_DI_01_Access_Reset AND (safeState[n] > 1) AND NOT masterReset[n]) THEN
//		//SafetyZone[n].Interlock.GS_DO_01_Lock_Solenoid := FALSE; //Reset after reset pressed and door shut
//		SafetyZone[n].AccessRequested := FALSE;
//		safeState[n] := 4; // Check zone status
//		//		ELSIF masterReset AND NOT SafetyZone[n].Zone_Status AND SafetyZone[n].ResetReady THEN
//		//			safeState[n] := 10; // Goto master reset state
//	END_IF;

	//Set disable to safe zone off or access requested
	SafetyZone[n].Disable := SafetyZone[n].AccessRequested OR NOT SafetyZone[n].Zone_Status;

	//-------------------------------------------------------
	//-------END--------Safety State Machine-------END-------
	//-------------------------------------------------------

	//-------------------------------------------------------
	//---------Set tower light status-&-TV-Indicators--------
	//-------------------------------------------------------
	IF (n > 0) THEN //Light tower 0 does not need to indicate access state.. It is used on the main cab to indicate alarms. See alarm Task.
		SafetyZone[n].TowerLight.TL_DO_Green := SafetyZone[n].TowerLight.TL_DO_Yellow := SafetyZone[n].TowerLight.TL_DO_Red := SafetyZone[n].TowerLight.TL_DO_Sounder := 0;
		CASE safeState[n] OF
			0: //Zone reset do not enter
				SafetyZone[n].TowerLight.TL_DO_Green 	:= SafetyZone[n].Zone_Status;
				SafetyZone[n].TowerLight.TL_DO_Red 		:= NOT SafetyZone[n].Zone_Status;
			1: //Access has been requested
				SafetyZone[n].TowerLight.TL_DO_Yellow 	:= Std.Clock1s; 	//Means Zone Ok but access requested
				SafetyZone[n].TowerLight.TL_DO_Green 	:= SafetyZone[n].Zone_Status;
				SafetyZone[n].TowerLight.TL_DO_Red 		:= NOT SafetyZone[n].Zone_Status;
			2: //Safe to enter no bags in transit and hoists in position
				SafetyZone[n].TowerLight.TL_DO_Yellow 	:= TRUE; //Amber & RED steady indicates safe to enter
				SafetyZone[n].TowerLight.TL_DO_Green 	:= SafetyZone[n].Zone_Status;
				SafetyZone[n].TowerLight.TL_DO_Red 		:= TRUE;
			3: //
				SafetyZone[n].TowerLight.TL_DO_Yellow 	:= Std.Clock200ms; //Amber/Green Alternate-- Enter with Caution
				SafetyZone[n].TowerLight.TL_DO_Sounder 	:= NOT ton_entryError[n].Q; //Short alarm to indicate enter with caution
				SafetyZone[n].TowerLight.TL_DO_Green 	:= NOT Std.Clock200ms;
			SafetyZone[n].TowerLight.TL_DO_Red 		:= NOT Std.Clock200ms OR SafetyZone[n].HoistsOutOfPosition; // If red ight on then fault

			4: //Ready for Reset
				SafetyZone[n].TowerLight.TL_DO_Yellow 	:= Std.Clock500ms AND SafetyZone[n].ResetReady; //Flash Yellow when ready to be reset
				SafetyZone[n].TowerLight.TL_DO_Green 	:= SafetyZone[n].Zone_Status;

			10://Master Reset Zone about to start
				SafetyZone[n].TowerLight.TL_DO_Sounder := TRUE;
				SafetyZone[n].TowerLight.TL_DO_Red := Std.Clock200ms; //Red fast flash indicates zone will reset

		END_CASE;

	END_IF;

	//-------------------------------------------------------------
	//-------END-Set tower light status-&-TV-Indicators-END--------
	//-------------------------------------------------------------

	//Check if the master reset has reset all zones.
	IF (masterReset[n] AND NOT SafetyZone[n].Zone_Status) THEN
		resetRequired := 1;
	END_IF;

	SafetyZone[n].Interlock.GS_DO_01_Lock_Solenoid := lockDoor[n];
	SafetyZone[n].LiftGates := (SafetyZone[n].Zone_Status AND (SafetyZone[n].BagsInTransit OR NOT SafetyZone[n].AccessRequested)); // Edge protection gates.

END_FOR;

IF NOT resetRequired THEN
	masterResetRequest := 0;
END_IF;
resetRequired := 0;

//Flash reset btn on main cabinet
IF masterResetRequest THEN // We can do a master reset and not out safe 0 to reset
	SafetyZone[0].Main_Lamp := Std.Clock200ms;
ELSE
	SafetyZone[0].Main_Lamp := Std.Clock1s AND NOT SafetyZone[0].Zone_Status;
END_IF;

//--------------------CUSTOMISTATION FOR INDICATION--------------------

//FOR n := 0 TO MAX_DUAL_CHANNELS DO
//	Indication[40 + n] := NOT SafetyZone[0].E_Stop.ES_SI_Two_Channel[n];
//END_FOR;
//
//Indication[61]	:= NOT SafetyZone[1].Interlock.GS_Two_Channel_Input;
//Indication[62]	:= NOT SafetyZone[2].Interlock.GS_Two_Channel_Input;
//Indication[63] 	:= NOT SafetyZone[3].Interlock.GS_Two_Channel_Input;
//Indication[64] 	:= NOT SafetyZone[4].Interlock.GS_Two_Channel_Input;
//
////Fire Doors
//Indication[65] 	:= NOT SafetyZone[1].E_Stop.ES_SI_Two_Channel[1];
//Indication[66] 	:= NOT SafetyZone[1].E_Stop.ES_SI_Two_Channel[2];

END_PROGRAM
```

#### Variables.var - Local variables
```iecst
VAR
	n : UINT;
	transitSettlePT : UDINT; (*Determines the amount of time to wait for bags in transit to settle before opening the interlock*)
	ton_10ms_Transit_Settle : ARRAY[0..MAX_SAFE_ZONES] OF TON_10ms; (*Determines the amount of time to wait for bags in transit to settle before opening the interlock*)
	safeState : ARRAY[0..MAX_SAFE_ZONES] OF USINT; (*USINT that tracks the state of the safe system so it can control the tower light*)
	debounceMasterPT : UDINT;
	masterReset : ARRAY[0..MAX_SAFE_ZONES] OF BOOL;
	ton_10ms_Master_Reset : TON_10ms;
	masterResetRequest : BOOL;
	startUpWarningPT : UDINT;
	ton_10ms_startUp_Warning : TON_10ms;
	tp_10ms_reset_Pulse : TP_10ms;
	enableMasterReset : BOOL;
	ton_10ms_Reset_Debounce : ARRAY[0..MAX_SAFE_ZONES] OF TON_10ms;
	ton_10ms_bagsInTransit : ARRAY[0..MAX_SAFE_ZONES] OF TON_10ms;
	f_trigRequestAccess : ARRAY[0..MAX_SAFE_ZONES] OF F_TRIG;
	ton_entryError : ARRAY[0..MAX_SAFE_ZONES] OF TON_10ms;
	resetRequired : BOOL;
	lockDoor : ARRAY[0..MAX_SAFE_ZONES] OF BOOL;
	tof_HoistsOutOfPosition : ARRAY[0..MAX_SAFE_ZONES] OF TOF_10ms;
END_VAR
```

### Program Logical/Safety/AccessControl (IEC) - *Mapping to allow access into zones

#### Main.st
```iecst
PROGRAM _CYCLIC

//	Std.SafetyOnZone[1]	;SPC1
//	Std.SafetyOnZone[2]	;SVC1
//	Std.SafetyOnZone[3]	;SVC2/3

//No access on zone 0

	SafetyZone[0].BagsInTransit :=  FALSE;  // Safe to enter when false (Switch is NO) FALSE WHEN OK..
	SafetyZone[0].HoistsOutOfPosition := FALSE; //<-- This is used to stop the door from opening if not position FALSE IS OK -- SWITCH IS NC..

	SafetyZone[1].BagsInTransit :=  FALSE;
	SafetyZone[1].HoistsOutOfPosition := FALSE;
//
	SafetyZone[2].BagsInTransit :=  FALSE;
	SafetyZone[2].HoistsOutOfPosition := Hoist_Safety[1].OutOfPosition;// OR Hoist_Safety[7].OutOfPosition;
//
	SafetyZone[3].BagsInTransit :=  FALSE;
	SafetyZone[3].HoistsOutOfPosition := FALSE;///Hoist_Safety[1].OutOfPosition OR Hoist_Safety[2].OutOfPosition OR Hoist_Safety[3].OutOfPosition;

END_PROGRAM
```

### Program Logical/Safety/SafetyUI (IEC) - Handling

#### SafetyUI.st - Implementation code
```iecst
(********************************************************************
* COPYRIGHT -- Bernecker + Rainer
********************************************************************
* Program: SafetySample
* File: SafetySample.st
* Author: B&R
********************************************************************
* Implementation of program SafetySample
********************************************************************)

PROGRAM _INIT

(* command structure for remote control FUB *)
	remotecmd.Version := safeVERSION_R107;	(* version *)
	remotecmd.Password := 'safeplc';				(* password *)
	remotecmd.NewPassword 	:= 'safeplc';

	remoteCmdGetStatus 		:= remotecmd;
	remoteCmdGetStatus.Command		:= safeCMD_STATUS;
	remoteCmdGetStatus.Data			:= 0;
	remoteCmdGetStatus.Number := 10;// ID to show request from auto refresh

	remoteControlcmd ACCESS ADR(remoteCmdGetStatus);

	(* command structure for application download *)
	appcmd1.Version := safeVERSION_R107;	(* version *)
	appcmd1.Password := 'safeplc';					(* password *)
	appcmd1.ApplicationID := 1;				(* application id *)

//	(* command structure for machine options download *)
//	datacmd1.Version := safeVERSION_R107;								(* version *)
//	datacmd1.Password := '';											(* password *)
//	datacmd1.pDeviceListInput := ADR(visuDeviceListInput);				(* device list *)
//	datacmd1.pMachineOptionsInput := ADR(dataMachineOptionsBitInput);	(* bit machine options *)
//	datacmd1.pModuleFlagsInput := ADR(dataModuleFlagsInput);			(* module flags *)
//	datacmd1.pAcknMachineOptions := ADR(dataAcknMachineOptions);		(* acknowledge information *)

//	(* command structure for extended machine options *)
//	datacmd2.Version := safeVERSION_R107;					(* version *)
//	datacmd2.Password := '';								(* password *)
//	datacmd2.pIntDataInput := ADR(visuIntInput);			(* INT channels *)
//	datacmd2.NumberIntInput := 1;							(* number of INT channels *)
//	datacmd2.pUintDataInput := ADR(visuUintInput);			(* UINT channels *)
//	datacmd2.NumberUintInput := 1;							(* number of UINT channels *)
//	datacmd2.pDintDataInput := ADR(visuDintInput);			(* DINT channels *)
//	datacmd2.NumberDintInput := 1;							(* number of DINT channels *)
//	datacmd2.pUdintDataInput := ADR(visuUdintInput);		(* UDINT channels *)
//	datacmd2.NumberUdintInput := 1;							(* number of UDINT channels *)
//	datacmd2.pAcknMachineOptions := ADR(visuAcknExtData);	(* acknowledge information *)

	(* hide elements in visualization *)
	FOR xcnt := 0 TO SIZEOF(statusButtonActiv) - 1 DO
		statusButtonActiv[xcnt] := 1;
	END_FOR

	(* hide elements in visualization *)
	statusButtonUnlockApp := 1;
	statusButtonUnlockData := 1;
	statusAcknInfoData := 1;
	statusButtonUnlockExtData := 1;
	statusAcknInfoExtData := 1;
	statusDialog := 1;

	(* set SafeLOGIC ID *)
	visuUsedSLIDRemote := 1;
	visuUsedSLIDData := 1;

	slxused := 1;
	safety := 0;
	visuEnableButtons := 0;

END_PROGRAM

PROGRAM _CYCLIC

//on init make sure we have set the password..

	ton_refreshStatus(IN := (safety > 0) AND SafetyPLC_Ok AND NOT safeRemoteControl_0.Busy AND NOT ton_refreshStatus.Q, PT:=100);

//	//Alarm for Hoist
//	IF (safeLogicStatus.SafeOSState <> 16#66) THEN //16# is Run[SAFE]
//		MpAlarmXSet(gAlarmXCore_Link,'SafetyPLCNotRunning');
//	ELSIF EDGEPOS(safeLogicStatus.SafeOSState = 16#66) THEN
//		MpAlarmXReset(gAlarmXCore_Link,'SafetyPLCNotRunning');
//	END_IF;
//	//End of Alarm

	CASE safety OF
		0: // Set the password on app load
			visuEnableButtons := 0;
			IF SafetyPLC_Ok THEN
				remotecmd.Command 	:= safeCMD_ENTER;
				remotecmd.Number 	:= 0;
				remotecmd.Data		:= safeCMD_SK_PW;
				IF safeRemoteControl_0.Done THEN
					safety := 10;
				ELSIF EDGEPOS(safeRemoteControl_0.Error) THEN
					execute := 0;
				END_IF;
				safeRemoteControl_0(SafeLOGICID := visuUsedSLIDRemote, Execute := execute, pCommandData := ADR(remotecmd));
				execute := 1;
			END_IF;

		10:// RUN UI

			//Lock the control buttons when the fub's are busy.
			visuEnableButtons := SafetyPLC_Ok AND ((remoteControlcmd.Number = 10) OR NOT safeRemoteControl_0.Busy) AND NOT safeDownloadApplication_0.Busy;
			(****************************************************************************************************************************************)
			(****************************************************************************************************************************************)
			(****************************************************************************************************************************************)
			(* show dialog to ackn command *)
			IF (dialogRemoteCmd = 1) THEN
				statusDialog := 0;
				dialogRemoteCmd := 0;
				indexButtonLeft := 0;
				indexButtonRight := 1;
				indexHeaderText := 0;
				IF (remotecmd.Data = safeCMD_SK_FORMAT) THEN
					indexMessageText := 0;
				ELSIF (remotecmd.Data = safeCMD_SK_XCHG) THEN
					indexMessageText := 1;
				ELSIF (remotecmd.Data = safeCMD_1_UDID_ACKN) THEN
					indexMessageText := 2;
				ELSIF (remotecmd.Data = safeCMD_2_UDID_ACKN) THEN
					indexMessageText := 3;
				ELSIF (remotecmd.Data = safeCMD_3_UDID_ACKN) THEN
					indexMessageText := 4;
				ELSIF (remotecmd.Data = safeCMD_4_UDID_ACKN) THEN
					indexMessageText := 5;
				ELSIF (remotecmd.Data =  safeCMD_N_UDID_ACKN) THEN
					indexMessageText := 6;
				ELSIF (remotecmd.Data =  safeCMD_CLEAR_DATA) THEN
					indexMessageText := 7;
				ELSIF (remotecmd.Data = safeCMD_FW_ACKN) THEN
					indexMessageText := 8;
				ELSIF (remotecmd.Data = safeCMD_RESET) THEN
					indexMessageText := 9;
				END_IF
			END_IF

			(* if dialog is ackn execute fub *)
			IF (dialogButtonLeft = 1 AND indexHeaderText = 0) THEN
				executeRemoteCmd := 1;
				dialogButtonLeft := 0;
				statusDialog := 1;
			ELSIF (dialogButtonRight = 1 AND indexHeaderText = 0) THEN
				dialogButtonRight := 0;
				statusDialog := 1;
			END_IF

			(* password must be at least 6 characters long *)
			IF brsstrlen(ADR(remotecmd.NewPassword)) < 6 THEN
				statusSetPassword := 2;
			ELSE
				statusSetPassword := 0;
			END_IF

			IF NOT safeRemoteControl_0.Busy THEN
				IF executeRemoteCmd THEN
					remoteControlcmd ACCESS ADR(remotecmd);
					executeRemoteControl := 1;
					executeRemoteCmd := 0;
				ELSIF ton_refreshStatus.Q THEN  // Set default, so we always read the status cyclically..
					executeRemoteControl := 1;
					remoteControlcmd ACCESS ADR(remoteCmdGetStatus);
				END_IF;
			END_IF;

			safeRemoteControl_0(SafeLOGICID := visuUsedSLIDRemote, Execute := executeRemoteControl, pCommandData := ADR(remoteControlcmd));
			executeRemoteControl := 0; // Make sure we always look at Rising edge inputs.

			(* reset execution flag *)
			IF (safeRemoteControl_0.Done = 1) THEN
				// If we have formatted or reset the key then wait for the PLC
				IF (remoteControlcmd.Data = safeCMD_CLEAR_DATA) OR (remoteControlcmd.Data = safeCMD_SK_FORMAT) THEN
					safety := 0;
				END_IF;
				safeLogicStatus := safeRemoteControl_0.SafeLOGICStatus;
			ELSIF (safeRemoteControl_0.Error = 1) THEN
				safety := 0;
			END_IF

			(* variables for visualization *)
			IF (safeLogicStatus.SafeKEYChanged = 1) THEN
				FOR xcnt := 0 TO SIZEOF(statusButtonActiv) - 1 DO
					statusButtonActiv[xcnt] := 1;
					statusButtonInactiv[xcnt] := 0;
				END_FOR
				statusButtonActiv[1] := 0;
				statusButtonInactiv[1] := 1;
			ELSIF (safeLogicStatus.NumberOfUDIDMismatches = 1 AND safeLogicStatus.Scanning = 0) THEN
				FOR xcnt := 0 TO SIZEOF(statusButtonActiv) - 1 DO
					statusButtonActiv[xcnt] := 1;
					statusButtonInactiv[xcnt] := 0;
				END_FOR
				statusButtonActiv[3] := 0;
				statusButtonInactiv[3] := 1;
			ELSIF (safeLogicStatus.NumberOfUDIDMismatches = 2 AND safeLogicStatus.Scanning = 0) THEN
				FOR xcnt := 0 TO SIZEOF(statusButtonActiv) - 1 DO
					statusButtonActiv[xcnt] := 1;
					statusButtonInactiv[xcnt] := 0;
				END_FOR
				statusButtonActiv[4] := 0;
				statusButtonInactiv[4] := 1;
			ELSIF (safeLogicStatus.NumberOfUDIDMismatches = 3 AND safeLogicStatus.Scanning = 0) THEN
				FOR xcnt := 0 TO SIZEOF(statusButtonActiv) - 1 DO
					statusButtonActiv[xcnt] := 1;
					statusButtonInactiv[xcnt] := 0;
				END_FOR
				statusButtonActiv[5] := 0;
				statusButtonInactiv[5] := 1;
			ELSIF (safeLogicStatus.NumberOfUDIDMismatches = 4 AND safeLogicStatus.Scanning = 0) THEN
				FOR xcnt := 0 TO SIZEOF(statusButtonActiv) - 1 DO
					statusButtonActiv[xcnt] := 1;
					statusButtonInactiv[xcnt] := 0;
				END_FOR
				statusButtonActiv[6] := 0;
				statusButtonInactiv[6] := 1;
			ELSIF (safeLogicStatus.NumberOfUDIDMismatches > 4 AND safeLogicStatus.Scanning = 0) THEN
				FOR xcnt := 0 TO SIZEOF(statusButtonActiv) - 1 DO
					statusButtonActiv[xcnt] := 1;
					statusButtonInactiv[xcnt] := 0;
				END_FOR
				statusButtonActiv[7] := 0;
				statusButtonInactiv[7] := 1;
			ELSIF (safeLogicStatus.NumberOfDifferentFirmware <> 0 AND safeLogicStatus.Scanning = 0) THEN
				FOR xcnt := 0 TO SIZEOF(statusButtonActiv) - 1 DO
					statusButtonActiv[xcnt] := 1;
					statusButtonInactiv[xcnt] := 0;
				END_FOR
				statusButtonActiv[11] := 0;
				statusButtonInactiv[11] := 1;
			ELSE
				FOR xcnt := 0 TO SIZEOF(statusButtonActiv) - 1 DO
					statusButtonActiv[xcnt] := 1;
					statusButtonInactiv[xcnt] := 0;
				END_FOR
			END_IF
			(* status text - MXCHG *)
			IF (safeLogicStatus.LedTestActive = 1) THEN
				indexMxchgLed := 40;
			ELSIF (safeLogicStatus.Scanning = 1) THEN
				indexMxchgLed := 30;
			ELSIF (safeLogicStatus.NumberOfUDIDMismatches = 1) THEN
				indexMxchgLed := 1;
			ELSIF (safeLogicStatus.NumberOfUDIDMismatches = 2) THEN
				indexMxchgLed := 2;
			ELSIF (safeLogicStatus.NumberOfUDIDMismatches = 3) THEN
				indexMxchgLed := 3;
			ELSIF (safeLogicStatus.NumberOfUDIDMismatches = 4) THEN
				indexMxchgLed := 4;
			ELSIF (safeLogicStatus.NumberOfUDIDMismatches > 4) THEN
				indexMxchgLed := 5;
			ELSIF (safeLogicStatus.NumberOfMissingModules <> 0) THEN
				indexMxchgLed := 20;
			ELSIF (safeLogicStatus.NumberOfUDIDMismatches = 0) THEN
				indexMxchgLed := 10;
			END_IF
			(* status text - FW-ACKN *)
			IF (safeLogicStatus.SafeKEYChanged = 0 AND safeLogicStatus.NumberOfDifferentFirmware = 0) THEN
				indexFwAcknLed := 10;
			ELSIF (safeLogicStatus.SafeKEYChanged = 1) THEN
				indexFwAcknLed := 1;
			ELSIF (safeLogicStatus.NumberOfDifferentFirmware <> 0) THEN
				indexFwAcknLed := 2;
			END_IF
			(* status text - FAIL *)
			IF (safeLogicStatus.FailSafe <> 16#55) THEN
				indexFAILLed := 2;
			ELSIF (safeLogicStatus.openSAFETYstate = 0) THEN
				indexFAILLed := 0;
			ELSIF (safeLogicStatus.openSAFETYstate = 1) THEN
				indexFAILLed := 1;
			END_IF
			(* status text - R/E *)
			indexRELed := safeLogicStatus.SafeOSState;

			(****************************************************************************************************************************************)
			(****************************************************************************************************************************************)
			(****************************************************************************************************************************************)
			(* show dialog to ackn command *)
			IF (dialogApplication = 1) THEN
				IF (statusDialog  <> 0) THEN
					statusDialog := 0;
					dialogApplication := 0;
					indexButtonLeft := 0;
					indexButtonRight := 1;
					indexHeaderText := 1;
					indexMessageText := 10;
				ELSE
					statusDialog := 1;
				END_IF;
			END_IF

			(* if dialog is ackn unlock application *)
			IF (dialogButtonLeft = 1 AND indexHeaderText = 1) THEN
				executeapp1 := 1;
				appcmd1.Unlock := 1;
				dialogButtonLeft := 0;
				statusDialog := 1;
			ELSIF (dialogButtonRight = 1 AND indexHeaderText = 1) THEN
				executeapp1 := 1;
				appcmd1.Unlock := 2;
				dialogButtonRight := 0;
				statusDialog := 1;
			END_IF

			(* convert application CRC to HEX string *)
			itoahex(safeDownloadApplication_0.ApplicationCRC, ADR(visuApplicationCRC));

			safeDownloadApplication_0(SafeLOGICID := appcmd1.ApplicationID, Execute := executeapp1, pCommandData := ADR(appcmd1));
			(* show unlock button *)
			IF (safeDownloadApplication_0.UnlockRequired = 1) THEN
				statusButtonUnlockApp := 0;
			ELSE
				appcmd1.Unlock := 0;
				statusButtonUnlockApp := 1;
			END_IF
			IF EDGEPOS(safeDownloadApplication_0.UnlockRequired = 1) THEN
				dialogApplication := 1;
			END_IF;

			IF (safeDownloadApplication_0.Done OR safeDownloadApplication_0.Error)  THEN
				executeapp1 := 0;
			END_IF;
//			(****************************************************************************************************************************************)
//			(****************************************************************************************************************************************)
//			(****************************************************************************************************************************************)
//			(* disable machine options *)
//			IF (visuEnableMachineOptions = FALSE) THEN
//				datacmd1.pMachineOptionsInput := 0;
//			ELSE
//				datacmd1.pMachineOptionsInput := ADR(dataMachineOptionsBitInput);
//			END_IF
//
//			(* disable module flags *)
//			IF (visuEnableModuleFlags = FALSE) THEN
//				datacmd1.pModuleFlagsInput := 0;
//			ELSE
//				datacmd1.pModuleFlagsInput := ADR(dataModuleFlagsInput);
//			END_IF
//
//			(* Machine Option Bit #000 *)
//			IF (visuMachineOptionsBitInput[0] = 1) THEN
//				dataMachineOptionsBitInput.BitData[0].0 := 1;
//			ELSE
//				dataMachineOptionsBitInput.BitData[0].0 := 0;
//			END_IF
//			(* Machine Option Bit #001 *)
//			IF (visuMachineOptionsBitInput[1] = 1) THEN
//				dataMachineOptionsBitInput.BitData[0].1 := 1;
//			ELSE
//				dataMachineOptionsBitInput.BitData[0].1 := 0;
//			END_IF
//			(* Machine Option Bit #002 *)
//			IF (visuMachineOptionsBitInput[2] = 1) THEN
//				dataMachineOptionsBitInput.BitData[0].2 := 1;
//			ELSE
//				dataMachineOptionsBitInput.BitData[0].2 := 0;
//			END_IF
//			(* Optional Flag Module #1 *)
//			IF (visuModuleFlagsOptionalInput[1] = 1) THEN
//				dataModuleFlagsInput.Optional[0].1 := 1;
//			ELSE
//				dataModuleFlagsInput.Optional[0].1 := 0;
//			END_IF
//			(* Optional Flag Module #2 *)
//			IF (visuModuleFlagsOptionalInput[2] = 1) THEN
//				dataModuleFlagsInput.Optional[0].2 := 1;
//			ELSE
//				dataModuleFlagsInput.Optional[0].2 := 0;
//			END_IF
//			(* Startup Flag Module #1 *)
//			IF (visuModuleFlagsStartupInput[1] = 1) THEN
//				dataModuleFlagsInput.Startup[0].1 := 1;
//			ELSE
//				dataModuleFlagsInput.Startup[0].1 := 0;
//			END_IF
//			(* Startup Flag Module #2 *)
//			IF (visuModuleFlagsStartupInput[2] = 1) THEN
//				dataModuleFlagsInput.Startup[0].2 := 1;
//			ELSE
//				dataModuleFlagsInput.Startup[0].2 := 0;
//			END_IF
//			(* Not_Present Flag Module #1 *)
//			IF (visuModuleFlagsNotPresentInput[1] = 1) THEN
//				dataModuleFlagsInput.NotPresent[0].1 := 1;
//			ELSE
//				dataModuleFlagsInput.NotPresent[0].1 := 0;
//			END_IF
//			(* Not_Present Flag Module #2 *)
//			IF (visuModuleFlagsNotPresentInput[2] = 1) THEN
//				dataModuleFlagsInput.NotPresent[0].2 := 1;
//			ELSE
//				dataModuleFlagsInput.NotPresent[0].2 := 0;
//			END_IF
//
//			(* Ackn Machine Option Bit #000 *)
//			IF (visuAcknMachineOptions[0] = 1) THEN
//				dataAcknMachineOptions.AcknBitOptions[0].0 := 1;
//			ELSE
//				dataAcknMachineOptions.AcknBitOptions[0].0 := 0;
//			END_IF
//			(* Ackn Machine Option Bit #001 *)
//			IF (visuAcknMachineOptions[1] = 1) THEN
//				dataAcknMachineOptions.AcknBitOptions[0].1 := 1;
//			ELSE
//				dataAcknMachineOptions.AcknBitOptions[0].1 := 0;
//			END_IF
//			(* Ackn Machine Option Bit #002 *)
//			IF (visuAcknMachineOptions[2] = 1) THEN
//				dataAcknMachineOptions.AcknBitOptions[0].2 := 1;
//			ELSE
//				dataAcknMachineOptions.AcknBitOptions[0].2 := 0;
//			END_IF
//
//			(* show dialog to ackn command *)
//			IF (dialogData = 1) THEN
//				statusDialog := 0;
//				dialogData := 0;
//				indexButtonLeft := 0;
//				indexButtonRight := 1;
//				indexHeaderText := 2;
//				indexMessageText := 11;
//			END_IF
//
//			(* if dialog is ackn unlock data *)
//			IF (dialogButtonLeft = 1 AND indexHeaderText = 2) THEN
//				datacmd1.Unlock := 1;
//				dialogButtonLeft := 0;
//				statusDialog := 1;
//			ELSIF (dialogButtonRight = 1 AND indexHeaderText = 2) THEN
//				datacmd1.Unlock := 2;
//				dialogButtonRight := 0;
//				statusDialog := 1;
//			END_IF

//			safeDownloadData_0(SafeLOGICID := visuUsedSLIDData, Execute := executedata1, Type:= safeDATA_TYPE_MAOP, pCommandData := ADR(datacmd1));
//
//			(* data compare failed *)
//			IF (safeDownloadData_0.StatusID = safeERR_DL_COMPARE_FAILED) THEN
//				indexCompareTextData := 2;
//			ELSE
//				indexCompareTextData := 0;
//			END_IF
//
//			IF (safeDownloadData_0.UnlockRequired = 1) THEN
//				(* data compare successful *)
//				indexCompareTextData := 1;
//				IF (datacmd1.pDeviceListOutput <> 0 AND datacmd1.NumberDevicesOutput <> 0) THEN
//					pDeviceListOut ACCESS datacmd1.pDeviceListOutput;
//
//					(* device #1 *)
//					visuDeviceListOutput[0].SADR := pDeviceListOut[0].SADR;
//					brsmemcpy(ADR(visuDeviceListOutput[0].UDID_High), ADR(pDeviceListOut[0].UDID[0]), 2);
//					(* swap UDID *)
//					visuDeviceListOutput[0].UDID_High := swapUINT(visuDeviceListOutput[0].UDID_High);
//					brsmemcpy(ADR(visuDeviceListOutput[0].UDID_Low), ADR(pDeviceListOut[0].UDID[2]), 4);
//					(* swap UDID *)
//					visuDeviceListOutput[0].UDID_Low := swapUDINT(visuDeviceListOutput[0].UDID_Low);
//					(* device #2 *)
//					visuDeviceListOutput[1].SADR := pDeviceListOut[1].SADR;
//					brsmemcpy(ADR(visuDeviceListOutput[1].UDID_High), ADR(pDeviceListOut[1].UDID[0]), 2);
//					(* swap UDID *)
//					visuDeviceListOutput[1].UDID_High := swapUINT(visuDeviceListOutput[1].UDID_High);
//					brsmemcpy(ADR(visuDeviceListOutput[1].UDID_Low), ADR(pDeviceListOut[1].UDID[2]), 4);
//					(* swap UDID *)
//					visuDeviceListOutput[1].UDID_Low := swapUDINT(visuDeviceListOutput[1].UDID_Low);
//				END_IF
//
//				IF (datacmd1.pMachineOptionsOutput <> 0) THEN
//					pMachineOptionsBitOut ACCESS datacmd1.pMachineOptionsOutput;
//
//					(* Machine Option Bit #000 *)
//					IF (pMachineOptionsBitOut.BitData[0].0 = 1) THEN
//						visuMachineOptionsBitOutput[0] := 1;
//					END_IF
//					(* Machine Option Bit #001 *)
//					IF (pMachineOptionsBitOut.BitData[0].1 = 1) THEN
//						visuMachineOptionsBitOutput[1] := 1;
//					END_IF
//					(* Machine Option Bit #002 *)
//					IF (pMachineOptionsBitOut.BitData[0].2 = 1) THEN
//						visuMachineOptionsBitOutput[2] := 1;
//					END_IF
//				END_IF
//
//				IF (datacmd1.pModuleFlagsOutput <> 0) THEN
//					pModuleFlagsOut ACCESS datacmd1.pModuleFlagsOutput;
//
//					(* Optional Flag Module #1 *)
//					IF (pModuleFlagsOut.Optional[0].1 = 1) THEN
//						visuModuleFlagsOptionalOutput[1] := 1;
//					END_IF
//					(* Optional Flag Module #2 *)
//					IF (pModuleFlagsOut.Optional[0].2 = 1) THEN
//						visuModuleFlagsOptionalOutput[2] := 1;
//					END_IF
//					(* Startup Flag Module #1 *)
//					IF (pModuleFlagsOut.Startup[0].1 = 1) THEN
//						visuModuleFlagsStartupOutput[1] := 1;
//					END_IF
//					(* Startup Flag Module #2 *)
//					IF (pModuleFlagsOut.Startup[0].2 = 1) THEN
//						visuModuleFlagsStartupOutput[2] := 1;
//					END_IF
//					(* Not_Present Flag Module #1 *)
//					IF (pModuleFlagsOut.NotPresent[0].1 = 1) THEN
//						visuModuleFlagsNotPresentOutput[1] := 1;
//					END_IF
//					(* Not_Present Flag Module #2 *)
//					IF (pModuleFlagsOut.NotPresent[0].2 = 1) THEN
//						visuModuleFlagsNotPresentOutput[2] := 1;
//					END_IF
//				END_IF
//				(* show ackn box *)
//				statusAcknInfoData := 0;
//				(* show unlock button unlocked if one ACK is set *)
//				IF (visuAcknMachineOptions[0] = 1 OR visuAcknMachineOptions[1] = 1 OR visuAcknMachineOptions[2] = 1) THEN
//					statusButtonUnlockData := 0;
//				END_IF
//			ELSIF (safeDownloadData_0.Done = 1 OR safeDownloadData_0.Error = 1) THEN
//				(* reset visualization elements *)
//				brsmemset(ADR(visuDeviceListOutput), 0, SIZEOF(visuDeviceListOutput));
//				brsmemset(ADR(visuMachineOptionsBitOutput), 0, SIZEOF(visuMachineOptionsBitOutput));
//				brsmemset(ADR(visuModuleFlagsOptionalOutput), 0, SIZEOF(visuModuleFlagsOptionalOutput));
//				brsmemset(ADR(visuModuleFlagsStartupOutput), 0, SIZEOF(visuModuleFlagsStartupOutput));
//				brsmemset(ADR(visuModuleFlagsNotPresentOutput), 0, SIZEOF(visuModuleFlagsNotPresentOutput));
//				(* hide ackn box *)
//				statusAcknInfoData := 1;
//				(* hide unlock button *)
//				datacmd1.Unlock := 0;
//				statusButtonUnlockData := 1;
//				(* reset ackn flags *)
//				visuAcknMachineOptions[0] := 0;
//				visuAcknMachineOptions[1] := 0;
//				visuAcknMachineOptions[2] := 0;
//			ELSE
//				(* hide ackn box *)
//				statusAcknInfoData := 1;
//				(* hide unlock button *)
//				datacmd1.Unlock := 0;
//				statusButtonUnlockData := 1;
//			END_IF

//			(****************************************************************************************************************************************)
//			(****************************************************************************************************************************************)
//			(****************************************************************************************************************************************)
//			(* Enable for INT set *)
//			IF (visuEnableINTOptions <> 0) THEN
//				datacmd2.pIntDataInput := ADR(visuIntInput);
//				datacmd2.NumberIntInput := 1;
//			ELSE
//				datacmd2.pIntDataInput := 0;
//				datacmd2.NumberIntInput := 0;
//			END_IF
//			(* Enable for UINT set *)
//			IF (visuEnableUINTOptions <> 0) THEN
//				datacmd2.pUintDataInput := ADR(visuUintInput);
//				datacmd2.NumberUintInput := 1;
//			ELSE
//				datacmd2.pUintDataInput := 0;
//				datacmd2.NumberUintInput := 0;
//			END_IF
//			(* Enable for DINT set *)
//			IF (visuEnableDINTOptions <> 0) THEN
//				datacmd2.pDintDataInput := ADR(visuDintInput);
//				datacmd2.NumberDintInput := 1;
//			ELSE
//				datacmd2.pDintDataInput := 0;
//				datacmd2.NumberDintInput := 0;
//			END_IF
//			(* Enable for UDINT set *)
//			IF (visuEnableUDINTOptions <> 0) THEN
//				datacmd2.pUdintDataInput := ADR(visuUdintInput);
//				datacmd2.NumberUdintInput := 1;
//			ELSE
//				datacmd2.pUdintDataInput := 0;
//				datacmd2.NumberUdintInput := 0;
//			END_IF
//
//			(* show dialog to ackn command *)
//			IF (dialogExtData = 1) THEN
//				statusDialog := 0;
//				dialogExtData := 0;
//				indexButtonLeft := 0;
//				indexButtonRight := 1;
//				indexHeaderText := 3;
//				indexMessageText := 11;
//			END_IF
//
//			(* if dialog is ackn unlock data *)
//			IF (dialogButtonLeft = 1 AND indexHeaderText = 3) THEN
//				datacmd2.Unlock := 1;
//				dialogButtonLeft := 0;
//				statusDialog := 1;
//			ELSIF (dialogButtonRight = 1 AND indexHeaderText = 3) THEN
//				datacmd2.Unlock := 2;
//				dialogButtonRight := 0;
//				statusDialog := 1;
//			END_IF
//
//			safeDownloadData_1(SafeLOGICID := visuUsedSLIDData, Execute := executedata2, Type:= safeDATA_TYPE_EXTMAOP, pCommandData := ADR(datacmd2));
//
//			(* data compare failed *)
//			IF (safeDownloadData_1.StatusID = safeERR_DL_COMPARE_FAILED) THEN
//				indexCompareTextExtData := 2;
//			ELSE
//				indexCompareTextExtData := 0;
//			END_IF
//
//			IF (safeDownloadData_1.UnlockRequired = 1) THEN
//				(* data compare successful *)
//				indexCompareTextExtData := 1;
//
//				(* INT channels *)
//				IF (datacmd2.pIntDataOutput <> 0 AND datacmd2.NumberIntOutput <> 0) THEN
//					brsmemcpy(ADR(visuIntOutput), datacmd2.pIntDataOutput, SIZEOF(visuIntOutput));
//				END_IF
//				(* UINT channels *)
//				IF (datacmd2.pUintDataOutput <> 0 AND datacmd2.NumberUintOutput <> 0) THEN
//					brsmemcpy(ADR(visuUintOutput), datacmd2.pUintDataOutput, SIZEOF(visuUintOutput));
//				END_IF
//				(* DINT channels *)
//				IF (datacmd2.pDintDataOutput <> 0 AND datacmd2.NumberDintOutput <> 0) THEN
//					brsmemcpy(ADR(visuDintOutput), datacmd2.pDintDataOutput, SIZEOF(visuDintOutput));
//				END_IF
//				(* UDINT channels *)
//				IF (datacmd2.pUdintDataOutput <> 0 AND datacmd2.NumberUdintOutput <> 0) THEN
//					brsmemcpy(ADR(visuUdintOutput), datacmd2.pUdintDataOutput, SIZEOF(visuUdintOutput));
//				END_IF
//				(* show ackn box *)
//				statusAcknInfoExtData := 0;
//				(* show unlock button if one ACK is set *)
//				IF (visuAcknExtData.AcknIntOptions[0] = 1 OR visuAcknExtData.AcknUintOptions[0] = 1 OR visuAcknExtData.AcknDintOptions[0] = 1 OR visuAcknExtData.AcknUdintOptions[0] = 1) THEN
//					statusButtonUnlockExtData := 0;
//				END_IF
//			ELSIF (safeDownloadData_1.Done = 1 OR safeDownloadData_1.Error = 1) THEN
//				(* reset visualization elements *)
//				brsmemset(ADR(visuIntOutput), 0, SIZEOF(visuIntOutput));
//				brsmemset(ADR(visuUintOutput), 0, SIZEOF(visuUintOutput));
//				brsmemset(ADR(visuDintOutput), 0, SIZEOF(visuDintOutput));
//				brsmemset(ADR(visuUdintOutput), 0, SIZEOF(visuUdintOutput));
//				(* hide ackn box *)
//				statusAcknInfoExtData := 1;
//				(* hide unlock button *)
//				datacmd2.Unlock := 0;
//				statusButtonUnlockExtData := 1;
//				(* reset ackn flags *)
//				visuAcknExtData.AcknIntOptions[0] := 0;
//				visuAcknExtData.AcknUintOptions[0] := 0;
//				visuAcknExtData.AcknDintOptions[0] := 0;
//				visuAcknExtData.AcknUdintOptions[0] := 0;
//			ELSE
//				(* hide ackn box *)
//				statusAcknInfoExtData := 1;
//				(* hide unlock button *)
//				datacmd2.Unlock := 0;
//				statusButtonUnlockExtData := 1;
//			END_IF

			(****************************************************************************************************************************************)
			(****************************************************************************************************************************************)
			(****************************************************************************************************************************************)
			(* read UDID from SafeLOGIC-X *)
			IF slxused = 1 THEN
				readUDIDlowSLX(enable := 1, pDeviceName := ADR(Station), pChannelName := ADR('UDID_low'));

				IF readUDIDlowSLX.status = 0 THEN
					UDID_Low := readUDIDlowSLX.value;
				ELSIF readUDIDlowSLX.status <> 65535 THEN
					UDID_Low := 0;
				END_IF

				readUDIDhighSLX(enable := 1, pDeviceName := ADR(Station), pChannelName := ADR('UDID_high'));

				IF readUDIDhighSLX.status = 0 THEN
					UDID_High := UDINT_TO_UINT(readUDIDhighSLX.value);
				ELSIF readUDIDhighSLX.status <> 65535 THEN
					UDID_High := 0;
				END_IF

				(* hide / show visualization elements *)
				stautsSLXInformation := 0;
				statusSLInformation := 1;
				(* read UDID form SafeLOGIC *)
			ELSE
				readUDIDlowSL(enable := 1, pDevice := ADR(Interface), node := Node, index := 16#2000, subindex := 6, pData := ADR(UDID_Low), datalen := SIZEOF(UDID_Low));

				IF readUDIDlowSL.status <> 0 AND readUDIDlowSL.status <> 65535 THEN
					UDID_Low := 0;
				END_IF

				readUDIDhighSL(enable := 1, pDevice := ADR(Interface), node := Node, index := 16#2000, subindex := 7, pData := ADR(UDID_High), datalen := SIZEOF(UDID_High));

				IF readUDIDhighSL.status <> 0 AND readUDIDhighSL.status <> 65535 THEN
					UDID_High := 0;
				END_IF

				(* hide / show visualization elements *)
				stautsSLXInformation := 1;
				statusSLInformation := 0;
			END_IF

	END_CASE;

	(* convert UDID to HEX string *)
	itoahex(UDID_Low, ADR(visuUDID_Low));
	itoahex(UDID_High, ADR(visuUDID_High));

	(****************************************************************************************************************************************)
	(****************************************************************************************************************************************)
	(****************************************************************************************************************************************)
	(* write UDID for SafeLOGIC to command structure *)
	appcmd1.UDID_Low := UDID_Low;
	appcmd1.UDID_High := UDID_High;
	datacmd1.UDID_Low := UDID_Low;
	datacmd1.UDID_High := UDID_High;
	datacmd2.UDID_Low := UDID_Low;
	datacmd2.UDID_High := UDID_High;

	(****************************************************************************************************************************************)
	(****************************************************************************************************************************************)
	(****************************************************************************************************************************************)
	(* mappView lists use strings for values rather than int,uint etc. convert UINT to Strings. *)
	strRE_Led := UINT_TO_STRING(indexRELed);
	strMXCHG_Led := UINT_TO_STRING(indexMxchgLed);
	strFWACKN_Led := UINT_TO_STRING(indexFwAcknLed);
	strFAIL_Led := UINT_TO_STRING(indexFAILLed);

	IF NOT SafetyPLC_Ok THEN
		strStatusID := '10';
	ELSIF (safety = 0) THEN
		IF (safeRemoteControl_0.StatusID = ERR_FUB_BUSY) THEN
			strStatusID := '11';
		ELSE
			strStatusID := UINT_TO_STRING(safeRemoteControl_0.StatusID);
		END_IF;
	ELSIF safeDownloadApplication_0.Busy OR safeDownloadApplication_0.Error  THEN
		strStatusID := UINT_TO_STRING(safeDownloadApplication_0.StatusID);
	ELSIF  ((safeRemoteControl_0.Busy AND remoteControlcmd.Number <> 10) OR safeRemoteControl_0.Error)  THEN
		strStatusID := UINT_TO_STRING(safeRemoteControl_0.StatusID);
	ELSE
		strStatusID := '1';//NOTHING
	END_IF;

	strStatus := UINT_TO_STRING(safeLogicStatus.Status);

	strDownloadStatus := UINT_TO_STRING(safeDownloadApplication_0.StatusID);
	//strDataStatus := UINT_TO_STRING(safeDownloadData_0.StatusID);
	strMessageTest := UINT_TO_STRING(indexMessageText);

	(* guide user by changing button to orange. *)
	IF (statusButtonActiv[0] = 1) THEN
		strSKFormatStyle := 'Kannegiesser1';
	ELSE
		strSKFormatStyle := 'orange';
	END_IF;

	IF (statusButtonActiv[1] = 1) THEN
		strSKXCHGtStyle := 'Kannegiesser1';
	ELSE
		strSKXCHGtStyle := 'orange';
	END_IF;

	IF (statusButtonActiv[2] = 1) THEN
		strScanStyle := 'Kannegiesser1';
	ELSE
		strScanStyle := 'orange';
	END_IF;

	IF (statusButtonActiv[3] = 1) THEN
		strAck1Style := 'Kannegiesser1';
	ELSE
		strAck1Style := 'orange';
	END_IF;

	IF (statusButtonActiv[4] = 1) THEN
		strAck2Style := 'Kannegiesser1';
	ELSE
		strAck2Style := 'orange';
	END_IF;

	IF (statusButtonActiv[5] = 1) THEN
		strAck3Style := 'Kannegiesser1';
	ELSE
		strAck3Style := 'orange';
	END_IF;

	IF (statusButtonActiv[6] = 1) THEN
		strAck4Style := 'Kannegiesser1';
	ELSE
		strAck4Style := 'orange';
	END_IF;

	IF (statusButtonActiv[7] = 1) THEN
		strAckNStyle := 'Kannegiesser1';
	ELSE
		strAckNStyle := 'orange';
	END_IF;

	IF (statusButtonActiv[8] = 1) THEN
		strClearStyle := 'Kannegiesser1';
	ELSE
		strClearStyle := 'orange';
	END_IF;

	IF (statusButtonActiv[9] = 1) THEN
		strTestStyle := 'Kannegiesser1';
	ELSE
		strTestStyle := 'orange';
	END_IF;

	IF (statusButtonActiv[11] = 1) THEN
		strFWACKNStyle := 'Kannegiesser1';
	ELSE
		strFWACKNStyle := 'orange';
	END_IF;

	IF (statusButtonUnlockApp = 0) THEN
		bVisAppButtons := TRUE;
	ELSE
		bVisAppButtons := FALSE;
	END_IF;

	IF (statusSLInformation = 0) THEN
		bVisInterfaceNode := TRUE;
		bVisStation := FALSE;
	ELSE
		bVisInterfaceNode := FALSE;
		bVisStation := TRUE;
	END_IF;

			END_PROGRAM
```

#### SafetyUI.var - Local variables
```iecst
(********************************************************************
 * COPYRIGHT -- Bernecker + Rainer
 ********************************************************************
 * Program: SafetySample
 * File: SafetySample.var
 * Author: B&R
 ********************************************************************
 * Local variables of program SafetySample
 ********************************************************************)
VAR
	appcmd1 : DownloadCmdApplicationTypeV1; (*command structure for application download*)
	dataAcknMachineOptions : DownloadAcknMaOpTypeV1; (*data to acknowledge bit machine options*)
	datacmd1 : DownloadCmdMaOpTypeV1; (*command structure for machine options download*)
	datacmd2 : DownloadCmdExtMaOpTypeV1; (*command structure for extended machine options download*)
	dataMachineOptionsBitInput : ConfigurationBitOptionsTypeV1; (*data for bit machine options*)
	dataModuleFlagsInput : ConfigurationModuleFlagsTypeV1; (*data for module flags*)
	dialogApplication : BOOL; (*visualization dialog for application download*)
	dialogButtonLeft : BOOL; (*left button in visualization dialog*)
	dialogButtonRight : BOOL; (*right button in visualization dialog*)
	dialogData : BOOL; (*visualization dialog for machine options download*)
	dialogExtData : BOOL; (*visualization dialog for extended machine options download*)
	dialogRemoteCmd : BOOL; (*visualization dialog for remote control*)
	executeapp1 : BOOL; (*execute application download*)
	executedata1 : BOOL; (*execute machine options download*)
	executedata2 : BOOL; (*execute extended machine options download*)
	executeRemoteCmd : BOOL; (*execute remote control*)
	indexButtonLeft : UINT; (*index for button text*)
	indexButtonRight : UINT; (* index for button text*)
	indexCompareTextData : UINT; (*index for compare message machine options*)
	indexCompareTextExtData : UINT; (*index for compare message extended machine options*)
	indexFAILLed : UINT; (*index FAIL led*)
	indexFwAcknLed : UINT; (*index FW-ACKN led*)
	indexHeaderText : UINT; (*index dialog header text*)
	indexMessageText : UINT; (*index message text*)
	indexMxchgLed : UINT; (*index MXCHG led*)
	indexRELed : UINT; (*index R/E led*)
	Interface : STRING[80] := 'IF3'; (*interface information for SafeLOGIC*)
	Node : USINT := 1; (*node information for SafeLOGIC*)
	pDeviceListOut : REFERENCE TO ARRAY[0..1] OF ConfigurationDeviceTypeV1; (*device list from FUB*)
	pMachineOptionsBitOut : REFERENCE TO ConfigurationBitOptionsTypeV1; (*bit machine options from FUB*)
	pModuleFlagsOut : REFERENCE TO ConfigurationModuleFlagsTypeV1; (*module flags form FUB*)
	readUDIDhighSL : EplSDORead; (*function block to read UDID high from device*)
	readUDIDhighSLX : AsIOAccRead; (*function block to read UDID high from device*)
	readUDIDlowSL : EplSDORead; (*function block to read UDID low from device*)
	readUDIDlowSLX : AsIOAccRead; (*function block to read UDID low from device*)
	remotecmd : RemoteControlCmdTypeV1; (*command structure for remote control*)
	safeDownloadApplication_0 : safeDownloadApplication; (*function block safeDownloadApplication*)
	safeDownloadData_0 : safeDownloadData; (*function block safeDownloadData*)
	safeDownloadData_1 : safeDownloadData; (*function block safeDownloadData*)
	safeRemoteControl_0 : safeRemoteControl; (*function block safeRemoteControl*)
	slxused : BOOL; (*SafeLOGIC-X is used*)
	Station : STRING[80] := 'IF6.ST1'; (*station information for SafeLOGIC-X*)
	statusAcknInfoData : UINT; (*acknowledge boxes for machine options*)
	statusAcknInfoExtData : UINT; (*acknowledge boxes for extended machine options*)
	statusButtonActiv : ARRAY[0..15] OF USINT; (*button activ*)
	statusButtonInactiv : ARRAY[0..15] OF USINT; (*button inactiv*)
	statusButtonUnlockApp : UINT; (*unlock buttons application*)
	statusButtonUnlockData : UINT; (*unlock buttons data*)
	statusButtonUnlockExtData : UINT; (*unlock buttons extended data*)
	statusDialog : UINT; (*dialog box*)
	statusSetPassword : UINT; (*visualization status to set password*)
	statusSLInformation : UINT; (*display information for SafeLOGIC*)
	stautsSLXInformation : UINT; (*display information for SafeLOGIC-X*)
	UDID_High : UINT; (*UDID_high for SafelOGIC*)
	UDID_Low : UDINT; (*UDID_low for SafeLOGIC*)
	visuAcknExtData : DownloadAcknExtMaOpTypeV1; (*acknowledge extended machine options*)
	visuAcknMachineOptions : ARRAY[0..511] OF BOOL; (*acknowledge machine options*)
	visuApplicationCRC : STRING[8]; (*CRC HEX string for visualization*)
	visuDeviceListInput : ARRAY[0..1] OF DownloadDeviceTypeV1; (*device list input*)
	visuDeviceListOutput : ARRAY[0..1] OF DownloadDeviceTypeV1; (*device list output*)
	visuDintInput : ConfigurationDintOptionsTypeV1; (*DINT channels input*)
	visuDintOutput : ConfigurationDintOptionsTypeV1; (*DINT channels output*)
	visuEnableDINTOptions : BOOL; (*enable DINT options*)
	visuEnableINTOptions : BOOL; (*enable INT options*)
	visuEnableMachineOptions : BOOL; (*enable BIT options*)
	visuEnableModuleFlags : BOOL; (*enable module flags*)
	visuEnableUDINTOptions : BOOL; (*enable UDINT options*)
	visuEnableUINTOptions : BOOL; (*enable UINT options*)
	visuIntInput : ConfigurationIntOptionsTypeV1; (*INT channels input*)
	visuIntOutput : ConfigurationIntOptionsTypeV1; (*INT channels output*)
	visuMachineOptionsBitInput : ARRAY[0..511] OF BOOL; (*BIT options input*)
	visuMachineOptionsBitOutput : ARRAY[0..511] OF BOOL; (*BIT options output*)
	visuModuleFlagsNotPresentInput : ARRAY[0..1023] OF BOOL; (*not present module flags input*)
	visuModuleFlagsNotPresentOutput : ARRAY[0..1023] OF BOOL; (*not present module flags output*)
	visuModuleFlagsOptionalInput : ARRAY[0..1023] OF BOOL; (*optional module flags input*)
	visuModuleFlagsOptionalOutput : ARRAY[0..1023] OF BOOL; (*optional module flags output*)
	visuModuleFlagsStartupInput : ARRAY[0..1023] OF BOOL; (*startup module flags input*)
	visuModuleFlagsStartupOutput : ARRAY[0..1023] OF BOOL; (*startup module flags output*)
	visuUDID_High : STRING[8]; (*UDID hex string for visualization*)
	visuUDID_Low : STRING[8]; (*UDID hex string for visualization*)
	visuUdintInput : ConfigurationUdintOptionsTypeV1; (*UDINT channels input*)
	visuUdintOutput : ConfigurationUdintOptionsTypeV1; (*UDINT channels output*)
	visuUintInput : ConfigurationUintOptionsTypeV1; (*UINT channels input*)
	visuUintOutput : ConfigurationUintOptionsTypeV1; (*UINT channels output*)
	visuUsedSLIDData : UINT; (*SafeLOGIC ID for data download*)
	visuUsedSLIDRemote : UINT; (*SafeLOGIC ID for remote control*)
	xcnt : UINT; (*counter variable*)
	strStatusID : STRING[10];
	strMXCHG_Led : STRING[10];
	strFWACKN_Led : STRING[10];
	strStatus : STRING[10];
	strRE_Led : STRING[10];
	strFAIL_Led : STRING[10];
	strMessageTest : STRING[10];
	bVisAppButtons : BOOL;
	bVisInterfaceNode : BOOL;
	bVisStation : BOOL;
	strDownloadStatus : STRING[10];
	strDataStatus : STRING[10];
	strSKFormatStyle : STRING[15];
	strSKXCHGtStyle : STRING[15];
	strScanStyle : STRING[15];
	strAck1Style : STRING[15];
	strAck2Style : STRING[15];
	strAck3Style : STRING[15];
	strAck4Style : STRING[15];
	strAckNStyle : STRING[15];
	strFWACKNStyle : STRING[15];
	strTestStyle : STRING[15];
	strClearStyle : STRING[15];
	safeLogicStatus : RemoteControlStatusTypeV1;
	visuEnableButtons : BOOL;
	safety : USINT;
	execute : BOOL;
	remoteControlcmd : REFERENCE TO RemoteControlCmdTypeV1;
	executeRemoteControl : BOOL;
	remoteCmdGetStatus : RemoteControlCmdTypeV1;
	ton_refreshStatus : TON_10ms;
END_VAR
```

### Hoist.typ - Local data types
```iecst
TYPE
	OpcUa_type : 	STRUCT
		VC : ARRAY[230..248]OF OpcUa_VC_type;
	END_STRUCT;
	OpcUa_VC_type : 	STRUCT
		Read : OpcUa_VC_Read_type;
		Write : OpcUa_VC_Write_type;
	END_STRUCT;
	OpcUa_VC_Write_type : 	STRUCT
		Heartbeat : BOOL;
		PermissionToMove : BOOL;
		TargetPosition : USINT;
		ReleaseBag : BOOL;
		ReceiveBag : BOOL;
		LoadBag : BOOL;
		BagInTransit : BOOL;
	END_STRUCT;
	OpcUa_VC_Read_type : 	STRUCT
		StatusInfo : STRING[80];
		ActPosition : REAL;
		PositionNo : USINT;
		ReleaseBag : BOOL;
		ReceiveBag : BOOL;
		Heartbeat : BOOL;
		ReadyToReceive : BOOL;
		Auto : BOOL;
		Manual : BOOL;
		Error : BOOL;
		ChuteBlocked : BOOL;
		BagOnCarriage : BOOL;
		IsHome : BOOL;
		Weight : DINT;
	END_STRUCT;
END_TYPE
```

### Program Logical/HoistLibrary/HoistServer (IEC)

#### Main.st - Init, cyclic, exit code
```iecst
PROGRAM _INIT

END_PROGRAM

PROGRAM _CYCLIC

	MTBasicsPWM_0.DutyCycle		:= 50;
	MTBasicsPWM_0.Period		:= 2;
	MTBasicsPWM_0.Enable		:= TRUE;
	MTBasicsPWM_0();

	CASE Std.PLCStn OF
		0:
			start := 230;
		1:
			start := 240;

		ELSE
			start := 10;
	END_CASE;

	FOR i := start TO start + 8 DO

		OpcUa.VC[i].Write.Heartbeat	:= MTBasicsPWM_0.Out;

		OpcUa.VC[i].Read.StatusInfo;
		OpcUa.VC[i].Read.ActPosition;
		OpcUa.VC[i].Read.PositionNo;
		OpcUa.VC[i].Read.ReceiveBag;
		OpcUa.VC[i].Read.ReleaseBag;
		OpcUa.VC[i].Read.Heartbeat;
		OpcUa.VC[i].Read.ReadyToReceive;

	END_FOR;

	(* Establish a connection to the client *)

(*	ReadHeartbeat;

	CASE Connect_to_OpcUaServer_step OF

		WAIT:

			IF Connect_OpcUa THEN

				Connect_to_OpcUaServer_step := CONNECT_TO_OPCUA;
			END_IF;

		CONNECT_TO_OPCUA:

			SessionConnectInfo_0.SecurityMsgMode := UASecurityMsgMode_None;
			SessionConnectInfo_0.SecurityPolicy := UASecurityPolicy_None;
			SessionConnectInfo_0.TransportProfile := UATP_UATcp;
			SessionConnectInfo_0.UserIdentityToken.UserIdentityTokenType := UAUITT_Anonymous;
			SessionConnectInfo_0.SessionTimeout := T#10m;
			SessionConnectInfo_0.MonitorConnection := T#10s;

			UA_Connect_0.ServerEndpointUrl := 'opc.tcp://10.44.10.244:4840';
			UA_Connect_0.Timeout := T#10s;
			UA_Connect_0.Execute := TRUE;
			UA_Connect_0.SessionConnectInfo := SessionConnectInfo_0;

			IF (UA_Connect_0.Done = 1) THEN
				UA_Connect_0.Execute := FALSE;
				Connect_OpcUa := FALSE;
				ConnectionHdl := UA_Connect_0.ConnectionHdl;
				Connect_to_OpcUaServer_step := GET_NAMESPACE;
			END_IF;

			IF (UA_Connect_0.Error = 1) THEN
				ConnectionHdl := 0;
				UA_Connect_0.Execute := FALSE;
				Connect_to_OpcUaServer_step := ERROR_OPCUA;
			END_IF;

		GET_NAMESPACE:

			UA_GetNamespaceIndex_0.ConnectionHdl := ConnectionHdl;
			UA_GetNamespaceIndex_0.NamespaceUri := 'urn:B&R/pv/';
			UA_GetNamespaceIndex_0.Timeout := T#5s;
			UA_GetNamespaceIndex_0.Execute := TRUE;

			IF (UA_GetNamespaceIndex_0.Done = 1) THEN
				NamespaceIndex := UA_GetNamespaceIndex_0.NamespaceIndex;
				UA_GetNamespaceIndex_0.Execute := FALSE;
				Connect_to_OpcUaServer_step := GET_NODE_HANDLE;
			END_IF;

			IF (UA_GetNamespaceIndex_0.Error = 1) THEN
				NamespaceIndex := 0;
				UA_GetNamespaceIndex_0.Execute := FALSE;
				Connect_to_OpcUaServer_step := ERROR_OPCUA;
			END_IF;

		GET_NODE_HANDLE:

			UANodeID_0[0].NamespaceIndex := NamespaceIndex;
			UANodeID_0[0].Identifier := '::Test_OpcUa_Client:WriteHeartbeat';
			UANodeID_0[0].IdentifierType := UAIdentifierType_String;

			UA_NodeGetHandleList_0.ConnectionHdl := ConnectionHdl;
			UA_NodeGetHandleList_0.NodeIDCount := 1;
			UA_NodeGetHandleList_0.NodeIDs := UANodeID_0;
			UA_NodeGetHandleList_0.Timeout := T#10s;
			UA_NodeGetHandleList_0.Execute := TRUE;

			IF (UA_NodeGetHandleList_0.Done = 1) THEN
				NodeHdls := UA_NodeGetHandleList_0.NodeHdls;
				UA_NodeGetHandleList_0.Execute := FALSE;
				Connect_to_OpcUaServer_step := READ_LIST;
			END_IF;

			IF (UA_NodeGetHandleList_0.Error = 1) THEN
				NodeHdls[0] := 0;

				UA_NodeGetHandleList_0.Execute := FALSE;
				Connect_to_OpcUaServer_step := ERROR_OPCUA;
			END_IF;

		READ_LIST:

			UANodeAdditionalInfo_0[0].AttributeId := UAAI_Value;
			UANodeAdditionalInfo_0[0].IndexRangeCount := 0;

			Variable_Rd0[0] := '::ServerTask:ReadHeartbeat';

			IF NOT UA_ReadList_0.Done THEN

				UA_ReadList_0
					(
					Execute := TRUE,
					ConnectionHdl := ConnectionHdl,
					NodeHdlCount := 1,
					NodeHdls := NodeHdls,
					NodeAddInfo := UANodeAdditionalInfo_0,
					Timeout := T#10s,
				Variables := Variable_Rd0);

				IF (UA_ReadList_0.Busy = 0) THEN
					UA_ReadList_0.Execute := FALSE;

					IF (UA_ReadList_0.Done = 1) THEN
						TimestampHeart := UA_ReadList_0.TimeStamps[0];

					END_IF;
					IF (UA_ReadList_0.Error = 1) THEN
						TimestampHeart := 0;
						Connect_to_OpcUaServer_step := ERROR_OPCUA;
					END_IF;
				END_IF;

			ELSIF StopReading THEN
				Connect_to_OpcUaServer_step := RELEASE_NODE;
				UA_ReadList_0.Execute := FALSE;

			ELSE
				UA_ReadList_0
					(
					Execute := FALSE,
					ConnectionHdl := ConnectionHdl,
					NodeHdlCount := 1,
					NodeHdls := NodeHdls,
					NodeAddInfo := UANodeAdditionalInfo_0,
					Timeout := T#10s,
				Variables := Variable_Rd0);
			END_IF;

		RELEASE_NODE:

			UA_NodeReleaseHandleList_0.ConnectionHdl := ConnectionHdl;
			UA_NodeReleaseHandleList_0.NodeHdlCount := 1;
			UA_NodeReleaseHandleList_0.NodeHdls := NodeHdls;
			UA_NodeReleaseHandleList_0.Timeout := T#10s;
			UA_NodeReleaseHandleList_0.Execute := TRUE;
			StopReading := FALSE;

			IF (UA_NodeReleaseHandleList_0.Done = 1) THEN
				NodeHdls[0] := 0;

				UA_NodeReleaseHandleList_0.Execute := FALSE;
				Connect_to_OpcUaServer_step := DISCONNECT_OPCUA;
			END_IF;

			IF (UA_NodeReleaseHandleList_0.Error = 1) THEN
				NodeHdls[0] := 0;

				UA_NodeReleaseHandleList_0.Execute := FALSE;
				Connect_to_OpcUaServer_step := ERROR_OPCUA;
			END_IF;

		DISCONNECT_OPCUA:

			UA_Disconnect_0.ConnectionHdl := ConnectionHdl;
			UA_Disconnect_0.Timeout := T#10s;
			UA_Disconnect_0.Execute := TRUE;

			IF (UA_Disconnect_0.Done = 1) THEN
				ConnectionHdl := 0;
				UA_Disconnect_0.Execute := FALSE;
				Connect_to_OpcUaServer_step := WAIT;
			END_IF;

			IF (UA_Disconnect_0.Error = 1) THEN
				ConnectionHdl := 0;
				UA_Disconnect_0.Execute := FALSE;
				Connect_to_OpcUaServer_step := ERROR_OPCUA;
			END_IF;

		ERROR_OPCUA:

	END_CASE;

	UA_Connect_0;
	UA_GetNamespaceIndex_0;
	UA_NodeGetHandleList_0;
	UA_NodeReleaseHandleList_0;
	UA_Disconnect_0;				*)

END_PROGRAM

PROGRAM _EXIT
	(* Insert code here *)

END_PROGRAM
```

#### Variables.var - Local variables
```iecst
(****************************************************)
VAR
	MTBasicsPWM_0 : MTBasicsPWM;
	i : USINT;
	pHmiOpcUa : REFERENCE TO OpcUa_VC_type;
	start : USINT;
END_VAR
```

- Visualisation Logical/mappView (not shown)

- FEPL-02_and_ACS380__1.hwi (not shown)

### Program Logical/ABB_EPL/Belt (IEC, version 1.00.1) - Belt base sequence

#### belt.st - Implementation code
```iecst
(********************************************************************
 * COPYRIGHT --
 ********************************************************************
 * Author: Stephen Healey
 * Created: July 02, 2018
 ********************************************************************)
//V1.00.1 First Release
PROGRAM _INIT
//Configuration
	mySeq							:= 0;	//Sequence number
	myIO							:= 0;
	myZone						:= 0;
	myBag							:= 0; //Buffer Bag
	myOutBag 					:= 0;
	myBelt						:= 1;
	drive							ACCESS ADR(ABB_EPL[myBelt].Cmd);
	status						ACCESS ADR(ABB_EPL[myBelt].Status);
	speedSlow					:= 30;
	speedFast					:= 60;
	drive.Acc_seconds := 0; //0 will default to 3 seconds
	drive.Dec_seconds := 0; //0 will default to 3 seconds
	drive.Direction		:= ABB_DIRECTION_FWD;
END_PROGRAM

PROGRAM _CYCLIC
//Inputs
I_BeltPhotocell := X[myIO].X01;

//Reset vars
O_RunBelt := FALSE;
O_RunSlow := FALSE;

//Alarm config
IF (myBag = 0) THEN
	Alarm[mySeq].Bag	:= mySeq + 10000;
ELSE
	Alarm[mySeq].Bag	:= myBag;
END_IF;

Alarm[mySeq].Name 		:= 0;
Alarm[mySeq].Beacon	:= TRUE;
Alarm[mySeq].Extra		:= 0;
Alarm[mySeq].Time		:= 3000;

//Setup Sequence
step := D[900 + mySeq];
//Setup Pulse contact
pls := (step <> lastStep);
lastStep := step;

//Sequence
IF (step = 0) THEN
	//Disabled
END_IF;

IF (step = 1) THEN
	//Run belt fast
	O_RunBelt := TRUE;
END_IF;

//Select target velocity
IF O_RunSlow THEN
	drive.TargetVelocity := speedSlow;
ELSE
	drive.TargetVelocity := speedFast;
END_IF;

//Belt Alarms
IF status.Tripped OR status.Warning OR NOT status.OnRemote THEN
	Alarm[mySeq].Name := ALM_INVERTOR_FAULT;
	Alarm[mySeq].Time		:= 5000;
END_IF;

//-----------------------------------
//PLC Outputs - adjust TO suit system
//-----------------------------------

drive.Run := O_RunBelt AND NOT Std.HaltSysZone[myZone];
drive.QuickStop := NOT Std.HaltSysZone[myZone];

//Alarms
timerAlarm(IN := NOT pls AND (Alarm[mySeq].Name > 0),PT:= Alarm[mySeq].Time);

Alarm[mySeq].On 	:= timerAlarm.Q;
Alarm[mySeq].ET 	:= timerAlarm.ET;

END_PROGRAM
```

#### belt.var - Local variables
```iecst
(********************************************************************
 * COPYRIGHT --
 ********************************************************************
 * Program: pr
 * File: pr.var
 * Author: treamsbottom
 * Created: July 16, 2015
 ********************************************************************
 * Local variables of program pr
 ********************************************************************)
VAR
	mySeq : UINT;
	myIO : UINT;
	myZone : UINT;
	myBag : UINT;
	step : UINT;
	pls : BOOL;
	timerAlarm : TON_10ms;
END_VAR
VAR RETAIN
	lastStep : UINT;
END_VAR
VAR
	myOutBag : UINT;
	myBelt : UINT;
	drive : REFERENCE TO ABB_EPL_cmd_typ;
	O_RunBelt : BOOL;
	O_RunSlow : BOOL;
	speedFast : INT;
	speedSlow : INT;
	status : REFERENCE TO ABB_EPL_status_typ;
	I_BeltPhotocell : BOOL;
END_VAR
```

### Program Logical/ABB_EPL/ABBSettings (IEC, version 1.00.1) - *APPLY Default settings to 

#### Main.st - Init, cyclic, exit code
```iecst
//V1.00.0 -- First Release
//V1.00.1 -- Correct scaling and add missing motor sizes

PROGRAM _INIT

	FOR n := 1 TO MAX_DRIVES DO
		ABB_EPL.Settings[n].Acc := 1;//50;
		ABB_EPL.Settings[n].Dec := 1;//30;
		ABB_EPL.Settings[n].Fast := 70;//60;
		ABB_EPL.Settings[n].Slow := 30;

		CASE ABB_EPL.Drives[n].Cmd.MotorSize OF // Need to set these values correctly

			ABB_MOTOR_0_25KW:
				ABB_EPL.Settings[n].MaxCurrent 		:= 190; //1.9A

			ABB_MOTOR_0_37KW_0_91A_1374:

				ABB_EPL.Settings[n].MaxCurrent 		:= 320; //3.2A

			ABB_MOTOR_0_37KW_0_97A_1342:
				ABB_EPL.Settings[n].MaxCurrent 		:= 350; //3.5A

			ABB_MOTOR_0_37KW_1_14A_1380:
				ABB_EPL.Settings[n].MaxCurrent 		:= 350;//3.5A

			ABB_MOTOR_0_75KW:
				ABB_EPL.Settings[n].MaxCurrent 		:= 1170; //11.7A

			ABB_MOTOR_1_5KW:
				ABB_EPL.Settings[n].MaxCurrent 		:= 2200; //22A ???

			ABB_MOTOR_2_2KW_4_75A_1450:
				ABB_EPL.Settings[n].MaxCurrent 		:= 3000; //30A ???

			ABB_MOTOR_3KW:
				ABB_EPL.Settings[n].MaxCurrent 		:= 5248; //52.48

			ABB_MOTOR_CUSTOM: // Future  Alow Motor data to be set individaully
				//ABB_EPL.Settings[n].MaxCurrent 		:= 5500;

		END_CASE;
	END_FOR;

END_PROGRAM

PROGRAM _CYCLIC

END_PROGRAM
```

#### Variables.var - Local variables
```iecst
VAR
	n : UINT;
END_VAR
```

### Program Logical/ABB_EPL/ABB_Driver (IEC, version 2.00.8)
